# B&R Automation Studio project NAELD004C00R10L518F00 (part 38)

#### Act_Background.st - Change By Project
```iecst
(** 2019-01-08 **)
ACTION Act_Background:

	//Resetting Physical Output
	memset(ADR(a_bPhysicalDO), 0, SIZEOF(a_bPhysicalDO));

	//Digital Output Mapping Physical Output With Config
	IF p_tyDOSettings.diSafetyRlyRst > 0 AND p_tyDOSettings.diSafetyRlyRst <= UDINT_TO_DINT(p_udiMax) THEN
		a_bPhysicalDO[p_tyDOSettings.diSafetyRlyRst]	:= p_bSafetyRlyRst;
	END_IF

	IF p_tyDOSettings.diTLRed > 0 AND p_tyDOSettings.diTLRed <= UDINT_TO_DINT(p_udiMax) THEN
		a_bPhysicalDO[p_tyDOSettings.diTLRed]	:= p_bTLRed;
	END_IF

	IF p_tyDOSettings.diTLAmber > 0 AND p_tyDOSettings.diTLAmber <= UDINT_TO_DINT(p_udiMax) THEN
		a_bPhysicalDO[p_tyDOSettings.diTLAmber]	:= p_bTLAmber;
	END_IF

	IF p_tyDOSettings.diTLGreen > 0 AND p_tyDOSettings.diTLGreen <= UDINT_TO_DINT(p_udiMax) THEN
		a_bPhysicalDO[p_tyDOSettings.diTLGreen]	:= p_bTLGreen;
	END_IF

	IF p_tyDOSettings.diBuzzer > 0 AND p_tyDOSettings.diBuzzer <= UDINT_TO_DINT(p_udiMax) THEN
		a_bPhysicalDO[p_tyDOSettings.diBuzzer]	:= p_bBuzzer;
	END_IF

	IF p_tyDOSettings.diDBAA > 0 AND p_tyDOSettings.diDBAA <= UDINT_TO_DINT(p_udiMax) THEN
		a_bPhysicalDO[p_tyDOSettings.diDBAA]	:= p_bDBAA;
	END_IF

	IF p_tyDOSettings.diDBAB > 0 AND p_tyDOSettings.diDBAB <= UDINT_TO_DINT(p_udiMax) THEN
		a_bPhysicalDO[p_tyDOSettings.diDBAB]	:= p_bDBAB;
	END_IF

	IF p_tyDOSettings.diPullerExtCtrl > 0 AND p_tyDOSettings.diPullerExtCtrl <= UDINT_TO_DINT(p_udiMax) THEN
		a_bPhysicalDO[p_tyDOSettings.diPullerExtCtrl]	:= p_bPullerExtCtrl;
	END_IF

	IF p_tyDOSettings.diPullerRetCtrl > 0 AND p_tyDOSettings.diPullerRetCtrl <= UDINT_TO_DINT(p_udiMax) THEN
		a_bPhysicalDO[p_tyDOSettings.diPullerRetCtrl]	:= p_bPullerRetCtrl;
	END_IF

	IF p_tyDOSettings.diRotPullerCtrl > 0 AND p_tyDOSettings.diRotPullerCtrl <= UDINT_TO_DINT(p_udiMax) THEN
		a_bPhysicalDO[p_tyDOSettings.diRotPullerCtrl]	:= p_bRotPullerCtrl;
	END_IF

	IF p_tyDOSettings.diMag1FixedClampCtrl > 0 AND p_tyDOSettings.diMag1FixedClampCtrl <= UDINT_TO_DINT(p_udiMax) THEN
		a_bPhysicalDO[p_tyDOSettings.diMag1FixedClampCtrl]	:= p_bMag1FixedClampCtrl;
	END_IF

	IF p_tyDOSettings.diMag1RemoteClampCtrl > 0 AND p_tyDOSettings.diMag1RemoteClampCtrl <= UDINT_TO_DINT(p_udiMax) THEN
		a_bPhysicalDO[p_tyDOSettings.diMag1RemoteClampCtrl]	:= p_bMag1RemoteClampCtrl;
	END_IF

	IF p_tyDOSettings.diMag2FixedClampCtrl > 0 AND p_tyDOSettings.diMag2FixedClampCtrl <= UDINT_TO_DINT(p_udiMax) THEN
		a_bPhysicalDO[p_tyDOSettings.diMag2FixedClampCtrl]	:= p_bMag2FixedClampCtrl;
	END_IF

	IF p_tyDOSettings.diMag2RemoteClampCtrl > 0 AND p_tyDOSettings.diMag2RemoteClampCtrl <= UDINT_TO_DINT(p_udiMax) THEN
		a_bPhysicalDO[p_tyDOSettings.diMag2RemoteClampCtrl]	:= p_bMag2RemoteClampCtrl;
	END_IF

	IF p_tyDOSettings.diMag3FixedClampCtrl > 0 AND p_tyDOSettings.diMag3FixedClampCtrl <= UDINT_TO_DINT(p_udiMax) THEN
		a_bPhysicalDO[p_tyDOSettings.diMag3FixedClampCtrl]	:= p_bMag3FixedClampCtrl;
	END_IF

	IF p_tyDOSettings.diMag3RemoteClampCtrl > 0 AND p_tyDOSettings.diMag3RemoteClampCtrl <= UDINT_TO_DINT(p_udiMax) THEN
		a_bPhysicalDO[p_tyDOSettings.diMag3RemoteClampCtrl]	:= p_bMag3RemoteClampCtrl;
	END_IF

	IF p_tyDOSettings.diMag4FixedClampCtrl > 0 AND p_tyDOSettings.diMag4FixedClampCtrl <= UDINT_TO_DINT(p_udiMax) THEN
		a_bPhysicalDO[p_tyDOSettings.diMag4FixedClampCtrl]	:= p_bMag4FixedClampCtrl;
	END_IF

	IF p_tyDOSettings.diMag4RemoteClampCtrl > 0 AND p_tyDOSettings.diMag4RemoteClampCtrl <= UDINT_TO_DINT(p_udiMax) THEN
		a_bPhysicalDO[p_tyDOSettings.diMag4RemoteClampCtrl]	:= p_bMag4RemoteClampCtrl;
	END_IF

		//open clamp control (new)
	IF p_tyDOSettings.diMag1FixedClampOpenCtrl > 0 AND p_tyDOSettings.diMag1FixedClampOpenCtrl <= UDINT_TO_DINT(p_udiMax) THEN
		a_bPhysicalDO[p_tyDOSettings.diMag1FixedClampOpenCtrl]	:= NOT p_bMag1FixedClampOpenCtrl;
	END_IF

	IF p_tyDOSettings.diMag1RemoteClampOpenCtrl > 0 AND p_tyDOSettings.diMag1RemoteClampOpenCtrl <= UDINT_TO_DINT(p_udiMax) THEN
		a_bPhysicalDO[p_tyDOSettings.diMag1RemoteClampOpenCtrl]	:= NOT p_bMag1RemoteClampOpenCtrl;
	END_IF

	IF p_tyDOSettings.diMag2FixedClampOpenCtrl > 0 AND p_tyDOSettings.diMag2FixedClampOpenCtrl <= UDINT_TO_DINT(p_udiMax) THEN
		a_bPhysicalDO[p_tyDOSettings.diMag2FixedClampOpenCtrl]	:= NOT p_bMag2FixedClampOpenCtrl;
	END_IF

	IF p_tyDOSettings.diMag2RemoteClampOpenCtrl > 0 AND p_tyDOSettings.diMag2RemoteClampOpenCtrl <= UDINT_TO_DINT(p_udiMax) THEN
		a_bPhysicalDO[p_tyDOSettings.diMag2RemoteClampOpenCtrl]	:= NOT p_bMag2RemoteClampOpenCtrl;
	END_IF

	IF p_tyDOSettings.diMag3FixedClampOpenCtrl > 0 AND p_tyDOSettings.diMag3FixedClampOpenCtrl <= UDINT_TO_DINT(p_udiMax) THEN
		a_bPhysicalDO[p_tyDOSettings.diMag3FixedClampOpenCtrl]	:= NOT p_bMag3FixedClampOpenCtrl;
	END_IF

	IF p_tyDOSettings.diMag3RemoteClampOpenCtrl > 0 AND p_tyDOSettings.diMag3RemoteClampOpenCtrl <= UDINT_TO_DINT(p_udiMax) THEN
		a_bPhysicalDO[p_tyDOSettings.diMag3RemoteClampOpenCtrl]	:= NOT p_bMag3RemoteClampOpenCtrl;
	END_IF

	IF bShutterTuning = FALSE THEN

		IF p_tyDOSettings.diInShutterOpenCtrl > 0 AND p_tyDOSettings.diInShutterOpenCtrl <= UDINT_TO_DINT(p_udiMax) THEN
			a_bPhysicalDO[p_tyDOSettings.diInShutterOpenCtrl]	:= p_bInShutterOpenCtrl;
		END_IF

		IF p_tyDOSettings.diInShutterCloseCtrl > 0 AND p_tyDOSettings.diInShutterCloseCtrl <= UDINT_TO_DINT(p_udiMax) THEN
			a_bPhysicalDO[p_tyDOSettings.diInShutterCloseCtrl]	:= p_bInShutterCloseCtrl;
		END_IF

		IF p_tyDOSettings.diInShutterOpenCtrl2 > 0 AND p_tyDOSettings.diInShutterOpenCtrl2 <= UDINT_TO_DINT(p_udiMax) THEN
			a_bPhysicalDO[p_tyDOSettings.diInShutterOpenCtrl2]	:= p_bInShutterOpenCtrl2;
		END_IF

		IF p_tyDOSettings.diInShutterCloseCtrl2 > 0 AND p_tyDOSettings.diInShutterCloseCtrl2 <= UDINT_TO_DINT(p_udiMax) THEN
			a_bPhysicalDO[p_tyDOSettings.diInShutterCloseCtrl2]	:= p_bInShutterCloseCtrl2;
		END_IF

		IF p_tyDOSettings.diInShutterOpenCtrl3 > 0 AND p_tyDOSettings.diInShutterOpenCtrl3 <= UDINT_TO_DINT(p_udiMax) THEN
			a_bPhysicalDO[p_tyDOSettings.diInShutterOpenCtrl3]	:= p_bInShutterOpenCtrl3;
		END_IF

		IF p_tyDOSettings.diInShutterCloseCtrl3 > 0 AND p_tyDOSettings.diInShutterCloseCtrl3 <= UDINT_TO_DINT(p_udiMax) THEN
			a_bPhysicalDO[p_tyDOSettings.diInShutterCloseCtrl3]	:= p_bInShutterCloseCtrl3;
		END_IF

		IF p_tyDOSettings.diOutShutterOpenCtrl > 0 AND p_tyDOSettings.diOutShutterOpenCtrl <= UDINT_TO_DINT(p_udiMax) THEN
			a_bPhysicalDO[p_tyDOSettings.diOutShutterOpenCtrl]	:= p_bOutShutterOpenCtrl;
		END_IF

		IF p_tyDOSettings.diOutShutterCloseCtrl > 0 AND p_tyDOSettings.diOutShutterCloseCtrl <= UDINT_TO_DINT(p_udiMax) THEN
			a_bPhysicalDO[p_tyDOSettings.diOutShutterCloseCtrl]	:= p_bOutShutterCloseCtrl;
		END_IF

		IF p_tyDOSettings.diOutShutterOpenCtrl2 > 0 AND p_tyDOSettings.diOutShutterOpenCtrl2 <= UDINT_TO_DINT(p_udiMax) THEN
			a_bPhysicalDO[p_tyDOSettings.diOutShutterOpenCtrl2]	:= p_bOutShutterOpenCtrl2;
		END_IF

		IF p_tyDOSettings.diOutShutterCloseCtrl2 > 0 AND p_tyDOSettings.diOutShutterCloseCtrl2 <= UDINT_TO_DINT(p_udiMax) THEN
			a_bPhysicalDO[p_tyDOSettings.diOutShutterCloseCtrl2]	:= p_bOutShutterCloseCtrl2;
		END_IF

	ELSE

		CASE usiShutterTuningStep OF
			0:
				a_bPhysicalDO[p_tyDOSettings.diInShutterOpenCtrl]	:= TRUE;
				a_bPhysicalDO[p_tyDOSettings.diOutShutterOpenCtrl]	:= TRUE;
				a_bPhysicalDO[p_tyDOSettings.diInShutterOpenCtrl2]	:= TRUE;
				a_bPhysicalDO[p_tyDOSettings.diInShutterOpenCtrl3]	:= TRUE;

				fbShutterTuneOpnTim(IN:= TRUE);
				IF fbShutterTuneOpnTim.Q THEN
					usiShutterTuningStep := 10;
					fbShutterTuneOpnTim(IN:= FALSE);
					a_bPhysicalDO[p_tyDOSettings.diInShutterOpenCtrl]	:= FALSE;
					a_bPhysicalDO[p_tyDOSettings.diOutShutterOpenCtrl]	:= FALSE;
					a_bPhysicalDO[p_tyDOSettings.diInShutterOpenCtrl2]	:= FALSE;
					a_bPhysicalDO[p_tyDOSettings.diInShutterOpenCtrl3]	:= FALSE;
				END_IF
			10:

				a_bPhysicalDO[p_tyDOSettings.diInShutterCloseCtrl]	:= TRUE;
				a_bPhysicalDO[p_tyDOSettings.diOutShutterCloseCtrl]	:= TRUE;
				a_bPhysicalDO[p_tyDOSettings.diInShutterCloseCtrl2]	:= TRUE;
				a_bPhysicalDO[p_tyDOSettings.diInShutterCloseCtrl3]	:= TRUE;

				fbShutterTuneClsTim(IN:= TRUE);
				IF fbShutterTuneClsTim.Q THEN
					usiShutterTuningStep := 0;
					fbShutterTuneClsTim(IN:= FALSE);
					a_bPhysicalDO[p_tyDOSettings.diInShutterCloseCtrl]	:= FALSE;
					a_bPhysicalDO[p_tyDOSettings.diOutShutterCloseCtrl]	:= FALSE;
					a_bPhysicalDO[p_tyDOSettings.diInShutterCloseCtrl2]	:= FALSE;
					a_bPhysicalDO[p_tyDOSettings.diInShutterCloseCtrl3]	:= FALSE;
				END_IF

		END_CASE
	END_IF

	IF p_tyDOSettings.diMag1ConvMtrIn > 0 AND p_tyDOSettings.diMag1ConvMtrIn <= UDINT_TO_DINT(p_udiMax) THEN
		a_bPhysicalDO[p_tyDOSettings.diMag1ConvMtrIn]	:= p_bMag1ConvMtrIn;
	END_IF

	IF p_tyDOSettings.diMag1ConvMtrOut > 0 AND p_tyDOSettings.diMag1ConvMtrOut <= UDINT_TO_DINT(p_udiMax) THEN
		a_bPhysicalDO[p_tyDOSettings.diMag1ConvMtrOut]	:= p_bMag1ConvMtrOut;
	END_IF

	IF p_tyDOSettings.diMag2ConvMtrIn > 0 AND p_tyDOSettings.diMag2ConvMtrIn <= UDINT_TO_DINT(p_udiMax) THEN
		a_bPhysicalDO[p_tyDOSettings.diMag2ConvMtrIn]	:= p_bMag2ConvMtrIn;
	END_IF

	IF p_tyDOSettings.diMag2ConvMtrOut > 0 AND p_tyDOSettings.diMag2ConvMtrOut <= UDINT_TO_DINT(p_udiMax) THEN
		a_bPhysicalDO[p_tyDOSettings.diMag2ConvMtrOut]	:= p_bMag2ConvMtrOut;
	END_IF

	IF p_tyDOSettings.diMag3ConvMtrIn > 0 AND p_tyDOSettings.diMag3ConvMtrIn <= UDINT_TO_DINT(p_udiMax) THEN
		a_bPhysicalDO[p_tyDOSettings.diMag3ConvMtrIn]	:= p_bMag3ConvMtrIn;
	END_IF

	IF p_tyDOSettings.diMag3ConvMtrOut > 0 AND p_tyDOSettings.diMag3ConvMtrOut <= UDINT_TO_DINT(p_udiMax) THEN
		a_bPhysicalDO[p_tyDOSettings.diMag3ConvMtrOut]	:= p_bMag3ConvMtrOut;
	END_IF

	IF p_tyDOSettings.diMag4ConvMtrIn > 0 AND p_tyDOSettings.diMag4ConvMtrIn <= UDINT_TO_DINT(p_udiMax) THEN
		a_bPhysicalDO[p_tyDOSettings.diMag4ConvMtrIn]	:= p_bMag4ConvMtrIn;
	END_IF

	IF p_tyDOSettings.diMag4ConvMtrOut > 0 AND p_tyDOSettings.diMag4ConvMtrOut <= UDINT_TO_DINT(p_udiMax) THEN
		a_bPhysicalDO[p_tyDOSettings.diMag4ConvMtrOut]	:= p_bMag4ConvMtrOut;
	END_IF

	IF p_tyDOSettings.diPullConvMtrOn > 0 AND p_tyDOSettings.diPullConvMtrOn <= UDINT_TO_DINT(p_udiMax) THEN
		a_bPhysicalDO[p_tyDOSettings.diPullConvMtrOn]	:= p_bPullConvMtrOn;
	END_IF

	IF p_tyDOSettings.diMag1SelClampCtrl > 0 AND p_tyDOSettings.diMag1SelClampCtrl <= UDINT_TO_DINT(p_udiMax) THEN
		a_bPhysicalDO[p_tyDOSettings.diMag1SelClampCtrl]	:= p_bMag1SelClampCtrl;
	END_IF

	IF p_tyDOSettings.diMag2SelClampCtrl > 0 AND p_tyDOSettings.diMag2SelClampCtrl <= UDINT_TO_DINT(p_udiMax) THEN
		a_bPhysicalDO[p_tyDOSettings.diMag2SelClampCtrl]	:= p_bMag2SelClampCtrl;
	END_IF

	IF p_tyDOSettings.diMag3SelClampCtrl > 0 AND p_tyDOSettings.diMag3SelClampCtrl <= UDINT_TO_DINT(p_udiMax) THEN
		a_bPhysicalDO[p_tyDOSettings.diMag3SelClampCtrl]	:= p_bMag3SelClampCtrl;
	END_IF

	IF p_tyDOSettings.diMag4SelClampCtrl > 0 AND p_tyDOSettings.diMag4SelClampCtrl <= UDINT_TO_DINT(p_udiMax) THEN
		a_bPhysicalDO[p_tyDOSettings.diMag4SelClampCtrl]	:= p_bMag4SelClampCtrl;
	END_IF

	IF bAgvComIODisabled = FALSE THEN
		//SOT Configuration
		IF p_tyDOSettings.diSOT1MagError > 0 AND p_tyDOSettings.diSOT1MagError <= UDINT_TO_DINT(p_udiMax) THEN
			a_bPhysicalDO[p_tyDOSettings.diSOT1MagError]				:= p_bSOTMagError1;
		END_IF

		IF p_tyDOSettings.diSOT1MagSizeLarge > 0 AND p_tyDOSettings.diSOT1MagSizeLarge <= UDINT_TO_DINT(p_udiMax) THEN
			a_bPhysicalDO[p_tyDOSettings.diSOT1MagSizeLarge]				:= p_bSOTMagSizeLarge1;
		END_IF

		IF p_tyDOSettings.diSOT1MagReady > 0 AND p_tyDOSettings.diSOT1MagReady <= UDINT_TO_DINT(p_udiMax) THEN
			a_bPhysicalDO[p_tyDOSettings.diSOT1MagReady]				:= p_bSOTMagReady1;
		END_IF

		IF p_tyDOSettings.diSOT1MagAvailable > 0 AND p_tyDOSettings.diSOT1MagAvailable <= UDINT_TO_DINT(p_udiMax) THEN
			a_bPhysicalDO[p_tyDOSettings.diSOT1MagAvailable]				:= p_bSOTMagAvailable1;
		END_IF

		IF p_tyDOSettings.diSOT2MagError > 0 AND p_tyDOSettings.diSOT2MagError <= UDINT_TO_DINT(p_udiMax) THEN
			a_bPhysicalDO[p_tyDOSettings.diSOT2MagError]				:= p_bSOTMagError2;
		END_IF

		IF p_tyDOSettings.diSOT2MagSizeLarge > 0 AND p_tyDOSettings.diSOT2MagSizeLarge <= UDINT_TO_DINT(p_udiMax) THEN
			a_bPhysicalDO[p_tyDOSettings.diSOT2MagSizeLarge]				:= p_bSOTMagSizeLarge2;
		END_IF

		IF p_tyDOSettings.diSOT2MagReady > 0 AND p_tyDOSettings.diSOT2MagReady <= UDINT_TO_DINT(p_udiMax) THEN
			a_bPhysicalDO[p_tyDOSettings.diSOT2MagReady]				:= p_bSOTMagReady2;
		END_IF

		IF p_tyDOSettings.diSOT2MagAvailable > 0 AND p_tyDOSettings.diSOT2MagAvailable <= UDINT_TO_DINT(p_udiMax) THEN
			a_bPhysicalDO[p_tyDOSettings.diSOT2MagAvailable]				:= p_bSOTMagAvailable2;
		END_IF

		IF p_tyDOSettings.diSOT3MagError > 0 AND p_tyDOSettings.diSOT3MagError <= UDINT_TO_DINT(p_udiMax) THEN
			a_bPhysicalDO[p_tyDOSettings.diSOT3MagError]				:= p_bSOTMagError3;
		END_IF

		IF p_tyDOSettings.diSOT3MagSizeLarge > 0 AND p_tyDOSettings.diSOT3MagSizeLarge <= UDINT_TO_DINT(p_udiMax) THEN
			a_bPhysicalDO[p_tyDOSettings.diSOT3MagSizeLarge]				:= p_bSOTMagSizeLarge3;
		END_IF

		IF p_tyDOSettings.diSOT3MagReady > 0 AND p_tyDOSettings.diSOT3MagReady <= UDINT_TO_DINT(p_udiMax) THEN
			a_bPhysicalDO[p_tyDOSettings.diSOT3MagReady]				:= p_bSOTMagReady3;
		END_IF

		IF p_tyDOSettings.diSOT3MagAvailable > 0 AND p_tyDOSettings.diSOT3MagAvailable <= UDINT_TO_DINT(p_udiMax) THEN
			a_bPhysicalDO[p_tyDOSettings.diSOT3MagAvailable]				:= p_bSOTMagAvailable3;
		END_IF

		IF p_tyDOSettings.diSOT4MagError > 0 AND p_tyDOSettings.diSOT4MagError <= UDINT_TO_DINT(p_udiMax) THEN
			a_bPhysicalDO[p_tyDOSettings.diSOT4MagError]				:= p_bSOTMagError4;
		END_IF

		IF p_tyDOSettings.diSOT4MagSizeLarge > 0 AND p_tyDOSettings.diSOT4MagSizeLarge <= UDINT_TO_DINT(p_udiMax) THEN
			a_bPhysicalDO[p_tyDOSettings.diSOT4MagSizeLarge]				:= p_bSOTMagSizeLarge4;
		END_IF

		IF p_tyDOSettings.diSOT4MagReady > 0 AND p_tyDOSettings.diSOT4MagReady <= UDINT_TO_DINT(p_udiMax) THEN
			a_bPhysicalDO[p_tyDOSettings.diSOT4MagReady]				:= p_bSOTMagReady4;
		END_IF

		IF p_tyDOSettings.diSOT4MagAvailable > 0 AND p_tyDOSettings.diSOT4MagAvailable <= UDINT_TO_DINT(p_udiMax) THEN
			a_bPhysicalDO[p_tyDOSettings.diSOT4MagAvailable]				:= p_bSOTMagAvailable4;
		END_IF

	ELSE
		a_bPhysicalDO[p_tyDOSettings.diSOT1MagError] := FALSE;
		a_bPhysicalDO[p_tyDOSettings.diSOT1MagSizeLarge] := FALSE;
		a_bPhysicalDO[p_tyDOSettings.diSOT1MagReady] := FALSE;
		a_bPhysicalDO[p_tyDOSettings.diSOT1MagAvailable] := FALSE;

		a_bPhysicalDO[p_tyDOSettings.diSOT2MagError] := FALSE;
		a_bPhysicalDO[p_tyDOSettings.diSOT2MagSizeLarge] := FALSE;
		a_bPhysicalDO[p_tyDOSettings.diSOT2MagReady] := FALSE;
		a_bPhysicalDO[p_tyDOSettings.diSOT2MagAvailable] := FALSE;

		a_bPhysicalDO[p_tyDOSettings.diSOT2MagError] := FALSE;
		a_bPhysicalDO[p_tyDOSettings.diSOT2MagSizeLarge] := FALSE;
		a_bPhysicalDO[p_tyDOSettings.diSOT2MagReady] := FALSE;
		a_bPhysicalDO[p_tyDOSettings.diSOT2MagAvailable] := FALSE;

		a_bPhysicalDO[p_tyDOSettings.diSOT2MagError] := FALSE;
		a_bPhysicalDO[p_tyDOSettings.diSOT2MagSizeLarge] := FALSE;
		a_bPhysicalDO[p_tyDOSettings.diSOT2MagReady] := FALSE;
		a_bPhysicalDO[p_tyDOSettings.diSOT2MagAvailable] := FALSE;
	END_IF

	IF p_eLinkAGVComProtocol = McSetAGVCommHardIO THEN
		IF p_tyDOSettings.diMag1ReqToBring > 0 AND p_tyDOSettings.diMag1ReqToBring <= UDINT_TO_DINT(p_udiMax) THEN
			a_bPhysicalDO[p_tyDOSettings.diMag1ReqToBring]				:= p_bRequestToBring1;
		END_IF

		IF p_tyDOSettings.diMag1ReqToGet > 0 AND p_tyDOSettings.diMag1ReqToGet <= UDINT_TO_DINT(p_udiMax) THEN
			a_bPhysicalDO[p_tyDOSettings.diMag1ReqToGet]				:= p_bRequestToGet1;
		END_IF

		IF p_tyDOSettings.diMag2ReqToBring > 0 AND p_tyDOSettings.diMag2ReqToBring <= UDINT_TO_DINT(p_udiMax) THEN
			a_bPhysicalDO[p_tyDOSettings.diMag2ReqToBring]				:= p_bRequestToBring2;
		END_IF

		IF p_tyDOSettings.diMag2ReqToGet > 0 AND p_tyDOSettings.diMag2ReqToGet <= UDINT_TO_DINT(p_udiMax) THEN
			a_bPhysicalDO[p_tyDOSettings.diMag2ReqToGet]				:= p_bRequestToGet2;
		END_IF

		IF p_tyDOSettings.diMag3ReqToBring > 0 AND p_tyDOSettings.diMag3ReqToBring <= UDINT_TO_DINT(p_udiMax) THEN
			a_bPhysicalDO[p_tyDOSettings.diMag3ReqToBring]				:= p_bRequestToBring3;
		END_IF

		IF p_tyDOSettings.diMag3ReqToGet > 0 AND p_tyDOSettings.diMag3ReqToGet <= UDINT_TO_DINT(p_udiMax) THEN
			a_bPhysicalDO[p_tyDOSettings.diMag3ReqToGet]				:= p_bRequestToGet3;
		END_IF

		IF p_tyDOSettings.diMag4ReqToBring > 0 AND p_tyDOSettings.diMag4ReqToBring <= UDINT_TO_DINT(p_udiMax) THEN
			a_bPhysicalDO[p_tyDOSettings.diMag4ReqToBring]				:= p_bRequestToBring4;
		END_IF

		IF p_tyDOSettings.diMag4ReqToGet > 0 AND p_tyDOSettings.diMag4ReqToGet <= UDINT_TO_DINT(p_udiMax) THEN
			a_bPhysicalDO[p_tyDOSettings.diMag4ReqToGet]				:= p_bRequestToGet4;
		END_IF
	ELSE
		a_bPhysicalDO[p_tyDOSettings.diMag1ReqToBring] := FALSE;
		a_bPhysicalDO[p_tyDOSettings.diMag1ReqToGet] := FALSE;
		a_bPhysicalDO[p_tyDOSettings.diMag2ReqToBring] := FALSE;
		a_bPhysicalDO[p_tyDOSettings.diMag2ReqToGet] := FALSE;
		a_bPhysicalDO[p_tyDOSettings.diMag3ReqToBring] := FALSE;
		a_bPhysicalDO[p_tyDOSettings.diMag3ReqToGet] := FALSE;
		a_bPhysicalDO[p_tyDOSettings.diMag4ReqToBring] := FALSE;
		a_bPhysicalDO[p_tyDOSettings.diMag4ReqToGet] := FALSE;
	END_IF

	IF p_tyDOSettings.diUSBRun > 0 AND p_tyDOSettings.diUSBRun <= UDINT_TO_DINT(p_udiMax) THEN
		a_bPhysicalDO[p_tyDOSettings.diUSBRun]	:= p_bUSBRun;
	END_IF

	IF p_tyDOSettings.diMtrPshrExt > 0 AND p_tyDOSettings.diMtrPshrExt <= UDINT_TO_DINT(p_udiMax) THEN
		a_bPhysicalDO[p_tyDOSettings.diMtrPshrExt]	:= p_bMtrPshrExt;
	END_IF

	IF p_tyDOSettings.diMtrPshrRet > 0 AND p_tyDOSettings.diMtrPshrRet <= UDINT_TO_DINT(p_udiMax) THEN
		a_bPhysicalDO[p_tyDOSettings.diMtrPshrRet]	:= p_bMtrPshrRet;
	END_IF

	IF p_tyDOSettings.diMtrPshrOn > 0 AND p_tyDOSettings.diMtrPshrOn <= UDINT_TO_DINT(p_udiMax) THEN
		a_bPhysicalDO[p_tyDOSettings.diMtrPshrOn]	:= p_bMtrPshrOn;
	END_IF

	IF p_tyDOSettings.diMtrPshrBrakeRls > 0 AND p_tyDOSettings.diMtrPshrBrakeRls <= UDINT_TO_DINT(p_udiMax) THEN
		a_bPhysicalDO[p_tyDOSettings.diMtrPshrBrakeRls]	:= p_bMtrPshrBrakeRls;
	END_IF

	IF p_tyDOSettings.diMtrPshrSpdBinBit0 > 0 AND p_tyDOSettings.diMtrPshrSpdBinBit0 <= UDINT_TO_DINT(p_udiMax) THEN
		a_bPhysicalDO[p_tyDOSettings.diMtrPshrSpdBinBit0]	:= p_bMtrPshrSpdBinBit0;
	END_IF

	IF p_tyDOSettings.diMtrPshrSpdBinBit1 > 0 AND p_tyDOSettings.diMtrPshrSpdBinBit1 <= UDINT_TO_DINT(p_udiMax) THEN
		a_bPhysicalDO[p_tyDOSettings.diMtrPshrSpdBinBit1]	:= p_bMtrPshrSpdBinBit1;
	END_IF

	IF p_tyDOSettings.diMtrPshrSpdBinBit2 > 0 AND p_tyDOSettings.diMtrPshrSpdBinBit2 <= UDINT_TO_DINT(p_udiMax) THEN
		a_bPhysicalDO[p_tyDOSettings.diMtrPshrSpdBinBit2]	:= p_bMtrPshrSpdBinBit2;
	END_IF

	IF p_tyDOSettings.diMtrPshrAlmRst > 0 AND p_tyDOSettings.diMtrPshrAlmRst <= UDINT_TO_DINT(p_udiMax) THEN
		a_bPhysicalDO[p_tyDOSettings.diMtrPshrAlmRst]	:= p_bMtrPshrAlmRst;
	END_IF

	IF p_tyDOSettings.diMag1SafetyBarRetCtrl > 0 AND p_tyDOSettings.diMag1SafetyBarRetCtrl <= UDINT_TO_DINT(p_udiMax) THEN
		a_bPhysicalDO[p_tyDOSettings.diMag1SafetyBarRetCtrl]	:= p_bMag1SafetyBarRetCtrl;
	END_IF

	IF p_tyDOSettings.diMag2SafetyBarRetCtrl > 0 AND p_tyDOSettings.diMag2SafetyBarRetCtrl <= UDINT_TO_DINT(p_udiMax) THEN
		a_bPhysicalDO[p_tyDOSettings.diMag2SafetyBarRetCtrl]	:= p_bMag2SafetyBarRetCtrl;
	END_IF

	IF p_tyDOSettings.diMag3SafetyBarRetCtrl > 0 AND p_tyDOSettings.diMag3SafetyBarRetCtrl <= UDINT_TO_DINT(p_udiMax) THEN
		a_bPhysicalDO[p_tyDOSettings.diMag3SafetyBarRetCtrl]	:= p_bMag3SafetyBarRetCtrl;
	END_IF

	IF p_tyDOSettings.diBypCurtainSen > 0 AND p_tyDOSettings.diBypCurtainSen <= UDINT_TO_DINT(p_udiMax) THEN
		a_bPhysicalDO[p_tyDOSettings.diBypCurtainSen]	:= p_bBypCurtainSen;
	END_IF

	IF p_tyDOSettings.diRstCurtainSen > 0 AND p_tyDOSettings.diRstCurtainSen <= UDINT_TO_DINT(p_udiMax) THEN
		a_bPhysicalDO[p_tyDOSettings.diRstCurtainSen]	:= p_bRstCurtainSen;
	END_IF

	IF p_tyDOSettings.diBypCurtainSensorPBLED > 0 AND p_tyDOSettings.diBypCurtainSensorPBLED <= UDINT_TO_DINT(p_udiMax) THEN	//JOHN
		a_bPhysicalDO[p_tyDOSettings.diBypCurtainSensorPBLED]	:= p_bBypCurtainPBLED;
	END_IF

	IF p_tyDOSettings.diMcSafetySigToDS > 0 AND p_tyDOSettings.diMcSafetySigToDS <= UDINT_TO_DINT(p_udiMax) THEN	//ADD
		a_bPhysicalDO[p_tyDOSettings.diMcSafetySigToDS]	:= p_bUIMachineSafetySigToDS;
	END_IF

	IF p_tyDOSettings.diTrolleyLckCtrl1 > 0 AND p_tyDOSettings.diTrolleyLckCtrl1 <= UDINT_TO_DINT(p_udiMax) THEN
		a_bPhysicalDO[p_tyDOSettings.diTrolleyLckCtrl1]	:= p_bTrolleyExtCtrl;
	END_IF
	IF p_tyDOSettings.diTrolleyLckCtrl2 > 0 AND p_tyDOSettings.diTrolleyLckCtrl2 <= UDINT_TO_DINT(p_udiMax) THEN
		a_bPhysicalDO[p_tyDOSettings.diTrolleyLckCtrl2]	:= p_bTrolleyExtCtrl2;
	END_IF

	//Update Output
	tyDOutput.bSafetyRlyRst			:= p_bSafetyRlyRst;
	tyDOutput.bTLRed				:= p_bTLRed;
	tyDOutput.bTLAmber				:= p_bTLAmber;
	tyDOutput.bTLGreen				:= p_bTLGreen;
	tyDOutput.bBuzzer				:= p_bBuzzer;
	tyDOutput.bDBAA					:= p_bDBAA;
	tyDOutput.bDBAB					:= p_bDBAB;
	tyDOutput.bPullerExtCtrl		:= p_bPullerExtCtrl;
	tyDOutput.bPullerRetCtrl		:= p_bPullerRetCtrl;
	tyDOutput.bRotPullerCtrl		:= p_bRotPullerCtrl;
	tyDOutput.bMag1FixedClampCtrl	:= p_bMag1FixedClampCtrl;
	tyDOutput.bMag1RemoteClampCtrl	:= p_bMag1RemoteClampCtrl;
	tyDOutput.bMag2FixedClampCtrl	:= p_bMag2FixedClampCtrl;
	tyDOutput.bMag2RemoteClampCtrl	:= p_bMag2RemoteClampCtrl;
	tyDOutput.bMag3FixedClampCtrl	:= p_bMag3FixedClampCtrl;
	tyDOutput.bMag3RemoteClampCtrl	:= p_bMag3RemoteClampCtrl;
	tyDOutput.bMag4FixedClampCtrl	:= p_bMag4FixedClampCtrl;
	tyDOutput.bMag4RemoteClampCtrl	:= p_bMag4RemoteClampCtrl;

	tyDOutput.bMag1FixedClampOpenCtrl  := p_bMag1FixedClampOpenCtrl; //new
	tyDOutput.bMag1RemoteClampOpenCtrl  := p_bMag1RemoteClampOpenCtrl;
	tyDOutput.bMag2FixedClampOpenCtrl  := p_bMag2FixedClampOpenCtrl;
	tyDOutput.bMag2RemoteClampOpenCtrl  := p_bMag2RemoteClampOpenCtrl;
	tyDOutput.bMag3FixedClampOpenCtrl  := p_bMag3FixedClampOpenCtrl;
	tyDOutput.bMag3RemoteClampOpenCtrl  := p_bMag3RemoteClampOpenCtrl;

	tyDOutput.bInShutterOpenCtrl	:= p_bInShutterOpenCtrl;
	tyDOutput.bInShutterCloseCtrl	:= p_bInShutterCloseCtrl;
	tyDOutput.bOutShutterOpenCtrl	:= p_bOutShutterOpenCtrl;
	tyDOutput.bOutShutterCloseCtrl	:= p_bOutShutterCloseCtrl;
	tyDOutput.bMag1ConvMtrIn		:= p_bMag1ConvMtrIn;
	tyDOutput.bMag1ConvMtrOut		:= p_bMag1ConvMtrOut;
	tyDOutput.bMag2ConvMtrIn		:= p_bMag2ConvMtrIn;
	tyDOutput.bMag2ConvMtrOut		:= p_bMag2ConvMtrOut;
	tyDOutput.bMag3ConvMtrIn		:= p_bMag3ConvMtrIn;
	tyDOutput.bMag3ConvMtrOut		:= p_bMag3ConvMtrOut;
	tyDOutput.bMag4ConvMtrIn		:= p_bMag4ConvMtrIn;
	tyDOutput.bMag4ConvMtrOut		:= p_bMag4ConvMtrOut;
	tyDOutput.bPullConvMtrOn		:= p_bPullConvMtrOn;
	tyDOutput.bMag1SelClampCtrl		:= p_bMag1SelClampCtrl;
	tyDOutput.bMag2SelClampCtrl		:= p_bMag2SelClampCtrl;
	tyDOutput.bMag3SelClampCtrl		:= p_bMag3SelClampCtrl;
	tyDOutput.bMag4SelClampCtrl		:= p_bMag4SelClampCtrl;
	tyDOutput.bSOT1MagAvailable		:= p_bSOTMagAvailable1;
	tyDOutput.bSOT2MagAvailable		:= p_bSOTMagAvailable2;
	tyDOutput.bSOT3MagAvailable		:= p_bSOTMagAvailable3;
	tyDOutput.bSOT4MagAvailable		:= p_bSOTMagAvailable4;
	tyDOutput.bSOT1MagError			:= p_bSOTMagError1;
	tyDOutput.bSOT2MagError			:= p_bSOTMagError2;
	tyDOutput.bSOT3MagError			:= p_bSOTMagError3;
	tyDOutput.bSOT4MagError			:= p_bSOTMagError4;
	tyDOutput.bSOT1MagReady			:= p_bSOTMagReady1;
	tyDOutput.bSOT2MagReady			:= p_bSOTMagReady2;
	tyDOutput.bSOT3MagReady			:= p_bSOTMagReady3;
	tyDOutput.bSOT4MagReady			:= p_bSOTMagReady4;
	tyDOutput.bSOT1MagSizeLarge		:= p_bSOTMagSizeLarge1;
	tyDOutput.bSOT2MagSizeLarge		:= p_bSOTMagSizeLarge2;
	tyDOutput.bSOT3MagSizeLarge		:= p_bSOTMagSizeLarge3;
	tyDOutput.bSOT4MagSizeLarge		:= p_bSOTMagSizeLarge4;
	tyDOutput.bMag1ReqToBring		:= a_bPhysicalDO[p_tyDOSettings.diMag1ReqToBring];
	tyDOutput.bMag1ReqToGet			:= a_bPhysicalDO[p_tyDOSettings.diMag1ReqToGet];
	tyDOutput.bMag2ReqToBring		:= a_bPhysicalDO[p_tyDOSettings.diMag2ReqToBring];
	tyDOutput.bMag2ReqToGet			:= a_bPhysicalDO[p_tyDOSettings.diMag2ReqToGet];
	tyDOutput.bMag3ReqToBring		:= a_bPhysicalDO[p_tyDOSettings.diMag3ReqToBring];
	tyDOutput.bMag3ReqToGet			:= a_bPhysicalDO[p_tyDOSettings.diMag3ReqToGet];
	tyDOutput.bMag4ReqToBring		:= a_bPhysicalDO[p_tyDOSettings.diMag4ReqToBring];
	tyDOutput.bMag4ReqToGet			:= a_bPhysicalDO[p_tyDOSettings.diMag4ReqToGet];
	tyDOutput.bUSBRun				:= p_bUSBRun;
	tyDOutput.bBypCurtainSen		:= p_bBypCurtainSen;
	tyDOutput.bRstCurtainSen		:= p_bRstCurtainSen;
	tyDOutput.bInShutterOpenCtrl2	:= p_bInShutterOpenCtrl2;
	tyDOutput.bInShutterCloseCtrl2	:= p_bInShutterCloseCtrl2;
	tyDOutput.bInShutterOpenCtrl3	:= p_bInShutterOpenCtrl3;
	tyDOutput.bInShutterCloseCtrl3	:= p_bInShutterCloseCtrl3;
	tyDOutput.bMcSafetySigToDS		:= p_bUIMachineSafetySigToDS;
	tyDOutput.bOutShutterOpenCtrl2	:= p_bOutShutterOpenCtrl2;
	tyDOutput.bOutShutterCloseCtrl2	:= p_bOutShutterCloseCtrl2;

END_ACTION
```

#### InputRef.var - Change By Project
```iecst
(*2019-05-20*)
(**)
(*General*)
VAR
	p_eAct : REFERENCE TO eDOAction;
	p_udiMax : REFERENCE TO UDINT;
END_VAR
(**)
(*Configuration*)
VAR
	p_tyDOSettings : REFERENCE TO tyDigitalOutputSettings;
END_VAR
(**)
VAR
	p_bManual : REFERENCE TO BOOL;
	p_bSafetyRlyRst : REFERENCE TO BOOL;
	p_bTLRed : REFERENCE TO BOOL;
	p_bTLAmber : REFERENCE TO BOOL;
	p_bTLGreen : REFERENCE TO BOOL;
	p_bBuzzer : REFERENCE TO BOOL;
	p_bDBAA : REFERENCE TO BOOL;
	p_bDBAB : REFERENCE TO BOOL;
	p_bPullerExtCtrl : REFERENCE TO BOOL;
	p_bPullerRetCtrl : REFERENCE TO BOOL;
	p_bRotPullerCtrl : REFERENCE TO BOOL;
	p_bMag1SelClampCtrl : REFERENCE TO BOOL;
	p_bMag2SelClampCtrl : REFERENCE TO BOOL;
	p_bMag3SelClampCtrl : REFERENCE TO BOOL;
	p_bMag4SelClampCtrl : REFERENCE TO BOOL;
	p_bMag1FixedClampCtrl : REFERENCE TO BOOL;
	p_bMag1RemoteClampCtrl : REFERENCE TO BOOL;
	p_bMag2FixedClampCtrl : REFERENCE TO BOOL;
	p_bMag2RemoteClampCtrl : REFERENCE TO BOOL;
	p_bMag3FixedClampCtrl : REFERENCE TO BOOL;
	p_bMag3RemoteClampCtrl : REFERENCE TO BOOL;
	p_bMag4FixedClampCtrl : REFERENCE TO BOOL;
	p_bMag4RemoteClampCtrl : REFERENCE TO BOOL;
	p_bInShutterOpenCtrl : REFERENCE TO BOOL;
	p_bInShutterOpenCtrl2 : REFERENCE TO BOOL;
	p_bInShutterOpenCtrl3 : REFERENCE TO BOOL;
	p_bInShutterCloseCtrl : REFERENCE TO BOOL;
	p_bInShutterCloseCtrl2 : REFERENCE TO BOOL;
	p_bInShutterCloseCtrl3 : REFERENCE TO BOOL;
	p_bOutShutterOpenCtrl : REFERENCE TO BOOL;
	p_bOutShutterCloseCtrl : REFERENCE TO BOOL;
	p_bOutShutterOpenCtrl2 : REFERENCE TO BOOL;
	p_bOutShutterCloseCtrl2 : REFERENCE TO BOOL;
	p_bMag1ConvMtrIn : REFERENCE TO BOOL;
	p_bMag1ConvMtrOut : REFERENCE TO BOOL;
	p_bMag2ConvMtrIn : REFERENCE TO BOOL;
	p_bMag2ConvMtrOut : REFERENCE TO BOOL;
	p_bMag3ConvMtrIn : REFERENCE TO BOOL;
	p_bMag3ConvMtrOut : REFERENCE TO BOOL;
	p_bMag4ConvMtrIn : REFERENCE TO BOOL;
	p_bMag4ConvMtrOut : REFERENCE TO BOOL;
	p_bPullConvMtrOn : REFERENCE TO BOOL;
	p_bSOTMagError1 : REFERENCE TO BOOL;
	p_bSOTMagSizeLarge1 : REFERENCE TO BOOL;
	p_bSOTMagReady1 : REFERENCE TO BOOL;
	p_bSOTMagAvailable1 : REFERENCE TO BOOL;
	p_bSOTMagError2 : REFERENCE TO BOOL;
	p_bSOTMagSizeLarge2 : REFERENCE TO BOOL;
	p_bSOTMagReady2 : REFERENCE TO BOOL;
	p_bSOTMagAvailable2 : REFERENCE TO BOOL;
	p_bSOTMagError3 : REFERENCE TO BOOL;
	p_bSOTMagSizeLarge3 : REFERENCE TO BOOL;
	p_bSOTMagReady3 : REFERENCE TO BOOL;
	p_bSOTMagAvailable3 : REFERENCE TO BOOL;
	p_bSOTMagError4 : REFERENCE TO BOOL;
	p_bSOTMagSizeLarge4 : REFERENCE TO BOOL;
	p_bSOTMagReady4 : REFERENCE TO BOOL;
	p_bSOTMagAvailable4 : REFERENCE TO BOOL;
	p_bUSBRun : REFERENCE TO BOOL;
	p_bMag1FixedClampOpenCtrl : REFERENCE TO BOOL;
	p_bMag1RemoteClampOpenCtrl : REFERENCE TO BOOL;
	p_bMag2FixedClampOpenCtrl : REFERENCE TO BOOL;
	p_bMag2RemoteClampOpenCtrl : REFERENCE TO BOOL;
	p_bMag3FixedClampOpenCtrl : REFERENCE TO BOOL;
	p_bMag3RemoteClampOpenCtrl : REFERENCE TO BOOL;
END_VAR
(**)
VAR
	p_bRequestToBring1 : REFERENCE TO BOOL;
	p_bRequestToBring2 : REFERENCE TO BOOL;
	p_bRequestToBring3 : REFERENCE TO BOOL;
	p_bRequestToBring4 : REFERENCE TO BOOL;
	p_bRequestToGet1 : REFERENCE TO BOOL;
	p_bRequestToGet2 : REFERENCE TO BOOL;
	p_bRequestToGet3 : REFERENCE TO BOOL;
	p_bRequestToGet4 : REFERENCE TO BOOL;
END_VAR
(**)
VAR
	p_bMtrPshrExt : REFERENCE TO BOOL;
	p_bMtrPshrRet : REFERENCE TO BOOL;
	p_bMtrPshrOn : REFERENCE TO BOOL;
	p_bMtrPshrBrakeRls : REFERENCE TO BOOL;
	p_bMtrPshrSpdBinBit0 : REFERENCE TO BOOL;
	p_bMtrPshrSpdBinBit1 : REFERENCE TO BOOL;
	p_bMtrPshrSpdBinBit2 : REFERENCE TO BOOL;
	p_bMtrPshrAlmRst : REFERENCE TO BOOL;
	p_bMag1SafetyBarRetCtrl : REFERENCE TO BOOL;
	p_bMag2SafetyBarRetCtrl : REFERENCE TO BOOL;
	p_bMag3SafetyBarRetCtrl : REFERENCE TO BOOL;
	p_bTrolleyExtCtrl : REFERENCE TO BOOL;
	p_bTrolleyExtCtrl2 : REFERENCE TO BOOL;
END_VAR
(**)
VAR
	p_bBypCurtainSen : REFERENCE TO BOOL;
	p_bRstCurtainSen : REFERENCE TO BOOL;
	p_bBypCurtainPBLED : REFERENCE TO BOOL;
	p_bUIMachineSafetySigToDS : REFERENCE TO BOOL;
	p_bDIDSUnlockSafetySig : REFERENCE TO BOOL;
END_VAR
```

#### Local.var - Change By Project
```iecst
(*2019-04-30*)
(**)
(*Local Action, State & Status*)
VAR
	eAct : eDOAction := DOActIdle;
	eStat : eDOAction := DOActIdle;
	eStatus : eFBStatus := Idle;
	sStatTxt : STRING[200] := '';
	a_sStatText : ARRAY[0..50] OF STRING[200] := ['Idling','Resetting All Special Output','Turning On Bypass Cover Switch','Turning Off Bypass Cover Switch',47('')];
END_VAR
(**)
(*Local Alarm*)
(**)
(*Local Output*)
VAR
	tyDOutput : tyDigitalOutput;
END_VAR
(**)
(*Local Input*)
VAR
	tyDOSettings : tyDigitalOutputSettings;
END_VAR
(**)
VAR
	bManual : BOOL := FALSE;
	bSafetyRlyRst : BOOL;
	bTLRed : BOOL;
	bTLAmber : BOOL;
	bTLGreen : BOOL;
	bBuzzer : BOOL;
	bDBAA : BOOL;
	bDBAB : BOOL;
	bPullerExtCtrl : BOOL;
	bPullerRetCtrl : BOOL;
	bRotPullerCtrl : BOOL;
	bMag1FixedClampCtrl : BOOL;
	bMag1RemoteClampCtrl : BOOL;
	bMag2FixedClampCtrl : BOOL;
	bMag2RemoteClampCtrl : BOOL;
	bMag3FixedClampCtrl : BOOL;
	bMag3RemoteClampCtrl : BOOL;
	bMag1FixedClampOpenCtrl : BOOL;
	bMag1RemoteClampOpenCtrl : BOOL;
	bMag2FixedClampOpenCtrl : BOOL;
	bMag2RemoteClampOpenCtrl : BOOL;
	bMag3FixedClampOpenCtrl : BOOL;
	bMag3RemoteClampOpenCtrl : BOOL;
	bInShutterOpenCtrl : BOOL;
	bInShutterCloseCtrl : BOOL;
	bOutShutterOpenCtrl : BOOL;
	bOutShutterCloseCtrl : BOOL;
	bMag1ConvMtrIn : BOOL;
	bMag1ConvMtrOut : BOOL;
	bMag2ConvMtrIn : BOOL;
	bMag2ConvMtrOut : BOOL;
	bMag3ConvMtrIn : BOOL;
	bMag3ConvMtrOut : BOOL;
	bPullConvMtrOn : BOOL;
	bMag1SelClampCtrl : BOOL;
	bMag2SelClampCtrl : BOOL;
	bMag3SelClampCtrl : BOOL;
	bSOTMagError1 : BOOL;
	bSOTMagSLarge1 : BOOL;
	bSOTMagReady1 : BOOL;
	bSOTMagAvailable1 : BOOL;
	bSOTMagError2 : BOOL;
	bSOTMagSLarge2 : BOOL;
	bSOTMagReady2 : BOOL;
	bSOTMagAvailable2 : BOOL;
	bSOTMagError3 : BOOL;
	bSOTMagSLarge3 : BOOL;
	bSOTMagReady3 : BOOL;
	bSOTMagAvailable3 : BOOL;
	bSOTMagError4 : BOOL;
	bSOTMagSLarge4 : BOOL;
	bSOTMagReady4 : BOOL;
	bSOTMagAvailable4 : BOOL;
	bRequestToBring1 : BOOL;
	bRequestToGet1 : BOOL;
	bRequestToBring2 : BOOL;
	bRequestToGet2 : BOOL;
	bRequestToBring3 : BOOL;
	bRequestToGet3 : BOOL;
	bRequestToBring4 : BOOL;
	bRequestToGet4 : BOOL;
	bMag1SafetyBarRetCtrl : BOOL;
	bMag2SafetyBarRetCtrl : BOOL;
	bMag3SafetyBarRetCtrl : BOOL;
	bBypCurtainPBLED : BOOL;
	bBypCurtainSen : BOOL;
	bRstCurtainSen : BOOL;
	bMcSafetySigDS : BOOL;
	bTrolleyExtCtrl : BOOL;
	bTrolleyExtCtrl2 : BOOL;
END_VAR
(**)
(*Local*)
VAR
	bInitDone : BOOL;
	bInitialDone : BOOL;
	a_bPhysicalDO : ARRAY[1..c_udiDOutputMax] OF BOOL;
	eStatOld : eDOAction := DOActIdle;
	usiShutterTuningStep : USINT := 0;
	bShutterTuning : BOOL;
	fbShutterTuneOpnTim : TON := (PT:=T#2s);
	fbShutterTuneClsTim : TON := (PT:=T#2s);
	bAgvComIODisabled : BOOL;
END_VAR
```

### Hermes.var - Change By Project
```iecst
(*2021-08-01*)
(**)
(*Action & State & Status*)
VAR
	p_HermesStat : UDINT;
	p_HermesStatus : UDINT;
	p_HermesStatTxt : UDINT;
	p_HermesMcParamAct : UDINT;
END_VAR
(**)
(*Alarm*)
VAR
	p_HermesAlmData : UDINT;
END_VAR
(**)
(*Output*)
VAR
	p_HermesFileNotFound : UDINT;
	p_HermesConfiguration : UDINT;
	p_HermesConfigurationWr : UDINT;
	p_HermesUSParam1 : UDINT;
	p_HermesUSParam2 : UDINT;
	p_HermesUSParam3 : UDINT;
	p_HermesUSParam4 : UDINT;
	p_HermesDSParam1 : UDINT;
	p_HermesDSParam2 : UDINT;
	p_HermesDSParam3 : UDINT;
	p_HermesDSParam4 : UDINT;
	p_HermesSvyParam : UDINT;
	p_HermesBrdAvlDataTable1stZ : UDINT;
	p_HermesBrdAvlDataTtlIdx1stZ : UDINT;
	p_HermesBrdAvlDataNewBrdAvl1stZ : UDINT;
	p_HermesBrdAvlDataTableLastZ : UDINT;
	p_HermesBrdAvlDataTtlIdxLastZ : UDINT;
	p_HermesBrdAvlDataNewBrdAvlLastZ : UDINT;
	p_HermesBrdId : UDINT;
END_VAR
```

### Program Logical/Hermes/Hermes (IEC) - 1.00.0 - NtHermes v5.00.0 , NtTCP v5.00.0 , NtMessage v5.00.0

#### InputRef.var
```iecst
(*2021-08-01*)
(**)
(*General*)
VAR
	p_eAct : REFERENCE TO eHermesAction;
	p_udiRstErr : REFERENCE TO UDINT;
	p_bPrep : REFERENCE TO BOOL;
	p_bEn : REFERENCE TO BOOL;
	p_bDis : REFERENCE TO BOOL;
END_VAR
(**)
(*Configuration*)
(**)
(*Input*)
VAR
	pa_tyUSParam : REFERENCE TO ARRAY[0..c_diHermesConfigMaxIdx] OF tyHermesUSParam;
	pa_tyDSParam : REFERENCE TO ARRAY[0..c_diHermesConfigMaxIdx] OF tyHermesDSParam;
	p_tyRmtParam : REFERENCE TO tyHermesRmtParam;
	p_tySvyParam : REFERENCE TO tyHermesSvyParam;
	p_sMcId : REFERENCE TO STRING[30];
	p_bRmtHermesWriteConfig : REFERENCE TO BOOL;
	p_bSvyHermesWriteConfig : REFERENCE TO BOOL;
	p_bUISaveHMIConfigure : REFERENCE TO BOOL;
	p_bUISaveHMISvyConfig : REFERENCE TO BOOL;
	p_tyRmtSetConfiguration : REFERENCE TO tyHermesCurrentConfiguration;
	p_bRmtPrep : REFERENCE TO BOOL;
	p_bRmtEn : REFERENCE TO BOOL;
	p_tySvySetConfiguration : REFERENCE TO tyHermesCurrentConfiguration;
	p_bSvyPrep : REFERENCE TO BOOL;
	p_bSvyEn : REFERENCE TO BOOL;
	p_sRetainFileName1 : REFERENCE TO STRING[80];
	p_sRetainFileName2 : REFERENCE TO STRING[80];
	p_sRetainFileName3 : REFERENCE TO STRING[80];
	p_sRetainFileName4 : REFERENCE TO STRING[80];
	p_udiRetainDataAddr1 : REFERENCE TO UDINT;
	p_udiRetainDataLen1 : REFERENCE TO UDINT;
	p_udiRetainDataAddr2 : REFERENCE TO UDINT;
	p_udiRetainDataLen2 : REFERENCE TO UDINT;
	p_udiRetainDataAddr3 : REFERENCE TO UDINT;
	p_udiRetainDataLen3 : REFERENCE TO UDINT;
	p_udiRetainDataAddr4 : REFERENCE TO UDINT;
	p_udiRetainDataLen4 : REFERENCE TO UDINT;
	p_sConfigFileName : REFERENCE TO STRING[80];
	p_sProgNm : REFERENCE TO STRING[15];
	p_bNtSettingsLoadDone : REFERENCE TO BOOL;
END_VAR
(**)
(*RmtHermes*)
VAR
	p_bRmtFoundIndexUS1 : REFERENCE TO BOOL;
	p_bRmtFoundIndexUS2 : REFERENCE TO BOOL;
	p_bRmtFoundIndexUS3 : REFERENCE TO BOOL;
	p_bRmtFoundIndexUS4 : REFERENCE TO BOOL;
	p_bRmtFoundIndexDS1 : REFERENCE TO BOOL;
	p_bRmtFoundIndexDS2 : REFERENCE TO BOOL;
	p_bRmtFoundIndexDS3 : REFERENCE TO BOOL;
	p_bRmtFoundIndexDS4 : REFERENCE TO BOOL;
	p_udiRmtIndexUS1 : REFERENCE TO UDINT;
	p_udiRmtIndexUS2 : REFERENCE TO UDINT;
	p_udiRmtIndexUS3 : REFERENCE TO UDINT;
	p_udiRmtIndexUS4 : REFERENCE TO UDINT;
	p_udiRmtIndexDS1 : REFERENCE TO UDINT;
	p_udiRmtIndexDS2 : REFERENCE TO UDINT;
	p_udiRmtIndexDS3 : REFERENCE TO UDINT;
	p_udiRmtIndexDS4 : REFERENCE TO UDINT;
END_VAR
(**)
(*SvyHermes*)
VAR
	p_bSvyFoundIndexUS1 : REFERENCE TO BOOL;
	p_bSvyFoundIndexUS2 : REFERENCE TO BOOL;
	p_bSvyFoundIndexUS3 : REFERENCE TO BOOL;
	p_bSvyFoundIndexUS4 : REFERENCE TO BOOL;
	p_bSvyFoundIndexDS1 : REFERENCE TO BOOL;
	p_bSvyFoundIndexDS2 : REFERENCE TO BOOL;
	p_bSvyFoundIndexDS3 : REFERENCE TO BOOL;
	p_bSvyFoundIndexDS4 : REFERENCE TO BOOL;
	p_udiSvyIndexUS1 : REFERENCE TO UDINT;
	p_udiSvyIndexUS2 : REFERENCE TO UDINT;
	p_udiSvyIndexUS3 : REFERENCE TO UDINT;
	p_udiSvyIndexUS4 : REFERENCE TO UDINT;
	p_udiSvyIndexDS1 : REFERENCE TO UDINT;
	p_udiSvyIndexDS2 : REFERENCE TO UDINT;
	p_udiSvyIndexDS3 : REFERENCE TO UDINT;
	p_udiSvyIndexDS4 : REFERENCE TO UDINT;
END_VAR
(**)
```

#### InputRef_Link.var
```iecst
(*2021-08-01*)
(**)
VAR
	p_bLinkStartupRun : REFERENCE TO BOOL;
	pa_usiMacAddr : REFERENCE TO ARRAY[0..5] OF USINT;
	p_tyDTStructure : REFERENCE TO DTStructure;
END_VAR
(**)
VAR
	pa_tyLinkXMLTableDataBrdAvl1 : REFERENCE TO ARRAY[0..200] OF tyXMLTableDat;
	p_iLinkXMLTableDataBrdAvlTtlIdx1 : REFERENCE TO INT;
	pa_tyLinkXMLTableDataBrdAvl2 : REFERENCE TO ARRAY[0..200] OF tyXMLTableDat;
	p_iLinkXMLTableDataBrdAvlTtlIdx2 : REFERENCE TO INT;
	pa_tyLinkXMLTableDataBrdAvl3 : REFERENCE TO ARRAY[0..200] OF tyXMLTableDat;
	p_iLinkXMLTableDataBrdAvlTtlIdx3 : REFERENCE TO INT;
	pa_tyLinkXMLTableDataBrdAvl4 : REFERENCE TO ARRAY[0..200] OF tyXMLTableDat;
	p_iLinkXMLTableDataBrdAvlTtlIdx4 : REFERENCE TO INT;
END_VAR
(**)
VAR
	tyHermesBrdAvlData : tyHermesBrdAvlDat;
	a_tyHermesBrdAvlData : ARRAY[1..200] OF tyHermesBrdAvlDat; (*Cater Up to 6 Zones*)
END_VAR
(**)
(*Zone 1*)
VAR
	p_bLinkOpsInitGConv1StepInitDone : REFERENCE TO BOOL;
	p_bLinkOpsInitGConv1MidHvBrd : REFERENCE TO BOOL;
	p_bLinkOpsInitGConv1EndHvBrd : REFERENCE TO BOOL;
	p_bLinkOpsGConv1HvBrd : REFERENCE TO BOOL;
	p_bLinkOpsGConv1StepEntBrd : REFERENCE TO BOOL;
	p_bLinkUSHermesTransporting : REFERENCE TO BOOL;
	p_bLinkUSSMEMATransporting : REFERENCE TO BOOL;
END_VAR
(**)
(*Zone 2*)
VAR
	p_bLinkOpsInitGConv2StepInitDone : REFERENCE TO BOOL;
	p_bLinkOpsInitGConv2MidHvBrd : REFERENCE TO BOOL;
	p_bLinkOpsInitGConv2EndHvBrd : REFERENCE TO BOOL;
	p_bLinkOpsGConv2HvBrd : REFERENCE TO BOOL;
	p_bLinkOpsGConv2StepEntBrd : REFERENCE TO BOOL;
	p_bLinkUSSMEMA2Transporting : REFERENCE TO BOOL;
END_VAR
(**)
```

#### Local.var
```iecst
(*2021-08-01*)
(**)
(*Local Action, State & Status*)
VAR
	eAct : eHermesAction := HermesActIdle;
	eStat : eHermesAction := HermesActIdle;
	eStatus : eFBStatus := Idle;
	udiStatus : UDINT := 0;
	sStatTxt : STRING[200] := '';
	a_sStatText : ARRAY[0..50] OF STRING[200] := ['Idling','Background Starting Operations','Background Stopping Operations','Deleting Old Log File','Creating Directory','Writing Retain File','Reading Retain File','Writing Configuration File','Reading Configuration File',42('')];
END_VAR
(**)
(*Local Alarm*)
VAR
	tyAlmData : tyAlmDat;
	a_tyAlmText : ARRAY[10000..10099] OF tyAlmTxt := [(sAlmText:='Create User Directory Error',sRcyText:='An Error Occurred While Attempting To Create User Directory. Please Contact Nutek For A Possible Solution'),(sAlmText:='Create Retain Directory Error',sRcyText:='An Error Occurred While Attempting To Create Retain Directory. Please Contact Nutek For A Possible Solution'),(sAlmText:='File Open Error While Reading Retain File',sRcyText:='An Error Was Encountered While Trying To Open File. Please Contact Nutek For A Possible Solution.'),(sAlmText:='File Read Error While Reading Retain File',sRcyText:='An Error Was Encountered While Trying To Read File. Please Contact Nutek For A Possible Solution.'),(sAlmText:='File Close Error While Reading Retain File',sRcyText:='An Error Was Encountered While Trying To Close File. Please Contact Nutek For A Possible Solution.'),(sAlmText:='File Open Error While Writing Retain File',sRcyText:='An Error Was Encountered While Trying To Open File. Please Contact Nutek For A Possible Solution.'),(sAlmText:='File Create Error While Writing Retain File',sRcyText:='An Error Was Encountered While Trying To Create File. Please Contact Nutek For A Possible Solution.'),(sAlmText:='File Write Error While Writing Retain File',sRcyText:='An Error Was Encountered While Trying To Write File. Please Contact Nutek For A Possible Solution.'),(sAlmText:='File Close Error While Writing Retain File',sRcyText:='An Error Was Encountered While Trying To Close File. Please Contact Nutek For A Possible Solution.'),(sAlmText:='Directory Does Not Exist While Writing Retain File',sRcyText:='The Directory Does Not Exist. Please Contact Nutek For A Possible Solution.'),(sAlmText:='Create Log Directory Error',sRcyText:='An Error Occurred While Attempting To Create Log Directory. Please Contact Nutek For A Possible Solution'),(sAlmText:='Create Machine Parameter Directory Error',sRcyText:='An Error Occurred While Attempting To Create Machine Parameter Directory. Please Contact Nutek For A Possible Solution'),(sAlmText:='File Open Error While Reading Config File',sRcyText:='An Error Was Encountered While Trying To Open File. Please Contact Nutek For A Possible Solution.'),(sAlmText:='File Read Error While Reading Config File',sRcyText:='An Error Was Encountered While Trying To Read File. Please Contact Nutek For A Possible Solution.'),(sAlmText:='File Close Error While Reading Config File',sRcyText:='An Error Was Encountered While Trying To Close File. Please Contact Nutek For A Possible Solution.'),(sAlmText:='File Open Error While Writing Config File',sRcyText:='An Error Was Encountered While Trying To Open File. Please Contact Nutek For A Possible Solution.'),(sAlmText:='File Create Error While Writing Config File',sRcyText:='An Error Was Encountered While Trying To Create File. Please Contact Nutek For A Possible Solution.'),(sAlmText:='File Write Error While Writing Config File',sRcyText:='An Error Was Encountered While Trying To Write File. Please Contact Nutek For A Possible Solution.'),(sAlmText:='File Close Error While Writing Config File',sRcyText:='An Error Was Encountered While Trying To Close File. Please Contact Nutek For A Possible Solution.'),(sAlmText:='Directory Does Not Exist While Writing Config File',sRcyText:='The Directory Does Not Exist. Please Contact Nutek For A Possible Solution.'),(0),2(0),3((0)),0,3((0)),(sAlmText:='File Open Error While Writing Retain File Lane 2',sRcyText:='An Error Was Encountered While Trying To Open File. Please Contact Nutek For A Possible Solution.'),(0),(sAlmText:='File Open Error While Reading Lane 2 Retain File',sRcyText:='An Error Was Encountered While Trying To Open File. Please Contact Nutek For A Possible Solution.'),(sAlmText:='File Read Error While Reading Lane 2 Retain File',sRcyText:='An Error Was Encountered While Trying To Read File. Please Contact Nutek For A Possible Solution.'),(sAlmText:='File Close Error While Reading Lane 2 Retain File',sRcyText:='An Error Was Encountered While Trying To Close File. Please Contact Nutek For A Possible Solution.'),(sAlmText:='File Open Error While Writing Lane 2 Retain File',sRcyText:='An Error Was Encountered While Trying To Open File. Please Contact Nutek For A Possible Solution.'),(sAlmText:='File Create Error While Writing Lane 2 Retain File',sRcyText:='An Error Was Encountered While Trying To Create File. Please Contact Nutek For A Possible Solution.'),(sAlmText:='File Write Error While Writing Lane 2 Retain File',sRcyText:='An Error Was Encountered While Trying To Write File. Please Contact Nutek For A Possible Solution.'),(sAlmText:='File Close Error While Writing Lane 2 Retain File',sRcyText:='An Error Was Encountered While Trying To Close File. Please Contact Nutek For A Possible Solution.'),(sAlmText:='Directory Does Not Exist While Writing Lane 2 Retain File',sRcyText:='The Directory Does Not Exist. Please Contact Nutek For A Possible Solution.'),2((0)),(sAlmText:='File Open Error While Reading Lane 3 Retain File',sRcyText:='An Error Was Encountered While Trying To Open File. Please Contact Nutek For A Possible Solution.'),(sAlmText:='File Read Error While Reading Lane 3 Retain File',sRcyText:='An Error Was Encountered While Trying To Read File. Please Contact Nutek For A Possible Solution.'),(sAlmText:='File Close Error While Reading Lane 3 Retain File',sRcyText:='An Error Was Encountered While Trying To Close File. Please Contact Nutek For A Possible Solution.'),(sAlmText:='File Open Error While Writing Lane 3 Retain File',sRcyText:='An Error Was Encountered While Trying To Open File. Please Contact Nutek For A Possible Solution.'),(sAlmText:='File Create Error While Writing Lane 3 Retain File',sRcyText:='An Error Was Encountered While Trying To Create File. Please Contact Nutek For A Possible Solution.'),(sAlmText:='File Write Error While Writing Lane 3 Retain File',sRcyText:='An Error Was Encountered While Trying To Write File. Please Contact Nutek For A Possible Solution.'),(sAlmText:='File Close Error While Writing Lane 3 Retain File',sRcyText:='An Error Was Encountered While Trying To Close File. Please Contact Nutek For A Possible Solution.'),(sAlmText:='Directory Does Not Exist While Writing Lane 3 Retain File',sRcyText:='The Directory Does Not Exist. Please Contact Nutek For A Possible Solution.'),2((0)),(sAlmText:='File Open Error While Reading Lane 4 Retain File',sRcyText:='An Error Was Encountered While Trying To Open File. Please Contact Nutek For A Possible Solution.'),(sAlmText:='File Read Error While Reading Lane 4 Retain File',sRcyText:='An Error Was Encountered While Trying To Read File. Please Contact Nutek For A Possible Solution.'),(sAlmText:='File Close Error While Reading Lane 4 Retain File',sRcyText:='An Error Was Encountered While Trying To Close File. Please Contact Nutek For A Possible Solution.'),(sAlmText:='File Open Error While Writing Lane 4 Retain File',sRcyText:='An Error Was Encountered While Trying To Open File. Please Contact Nutek For A Possible Solution.'),(sAlmText:='File Create Error While Writing Lane 4 Retain File',sRcyText:='An Error Was Encountered While Trying To Create File. Please Contact Nutek For A Possible Solution.'),(sAlmText:='File Write Error While Writing Lane 4 Retain File',sRcyText:='An Error Was Encountered While Trying To Write File. Please Contact Nutek For A Possible Solution.'),(sAlmText:='File Close Error While Writing Lane 4 Retain File',sRcyText:='An Error Was Encountered While Trying To Close File. Please Contact Nutek For A Possible Solution.'),(sAlmText:='Directory Does Not Exist While Writing Lane 4 Retain File',sRcyText:='The Directory Does Not Exist. Please Contact Nutek For A Possible Solution.'),40((0))];
END_VAR
(**)
(*Local Output*)
VAR
	bFileNotFound : BOOL;
	tyCurrConfiguration : tyHermesConfiguration := (a_tyUSParam:=[(tSndAlive:=T#60s,iLaneID:=1),3(0)],a_tyDSParam:=[(tSndAlive:=T#60s,uiSvrPort:=502,iLaneID:=1),0,2((0))]);
	tyConfigurationWr : tyHermesConfiguration;
END_VAR
(**)
(*Local Input*)
VAR
	udiRstErr : UDINT := 0;
	bPrep : BOOL := TRUE;
	bEn : BOOL := TRUE;
	bDis : BOOL := FALSE;
	a_tyUSParam : ARRAY[0..c_diHermesConfigMaxIdx] OF tyHermesUSParam;
	a_tyDSParam : ARRAY[0..c_diHermesConfigMaxIdx] OF tyHermesDSParam;
	tyRmtParam : tyHermesRmtParam;
	tySvyParam : tyHermesSvyParam;
	tyRmtSetConfiguration : tyHermesCurrentConfiguration;
	tySvySetConfiguration : tyHermesCurrentConfiguration;
	bRmtPrep : BOOL := FALSE;
	bRmtEn : BOOL := FALSE;
	bSvyPrep : BOOL := FALSE;
	bSvyEn : BOOL := FALSE;
	sRetainFileName1 : STRING[80] := 'HermesLane1.dat';
	sRetainFileName2 : STRING[80] := 'HermesLane2.dat';
	sRetainFileName3 : STRING[80] := 'HermesLane3.dat';
	sRetainFileName4 : STRING[80] := 'HermesLane4.dat';
	udiRetainDataAddr1 : UDINT;
	udiRetainDataLen1 : UDINT;
	udiRetainDataAddr2 : UDINT;
	udiRetainDataLen2 : UDINT;
	udiRetainDataAddr3 : UDINT;
	udiRetainDataLen3 : UDINT;
	udiRetainDataAddr4 : UDINT;
	udiRetainDataLen4 : UDINT;
	sConfigFileName : STRING[80] := 'Hermes.dat';
	sProgNm : STRING[15] := 'Hermes';
	bNtSettingsLoadDone : BOOL := TRUE;
	bRmtHermesWriteConfig : BOOL := TRUE;
	bSvyHermesWriteConfig : BOOL := TRUE;
	bUISaveHMIConfigure : BOOL := TRUE;
	bUISaveHMISvyConfig : BOOL := TRUE;
	sMcId : STRING[30] := '';
	bRmtFoundIndexUS1 : BOOL := FALSE;
	bRmtFoundIndexUS2 : BOOL := FALSE;
	bRmtFoundIndexUS3 : BOOL := FALSE;
	bRmtFoundIndexUS4 : BOOL := FALSE;
	bRmtFoundIndexDS1 : BOOL := FALSE;
	bRmtFoundIndexDS2 : BOOL := FALSE;
	bRmtFoundIndexDS3 : BOOL := FALSE;
	bRmtFoundIndexDS4 : BOOL := FALSE;
	udiRmtIndexUS1 : UDINT := 0;
	udiRmtIndexUS2 : UDINT := 0;
	udiRmtIndexUS3 : UDINT := 0;
	udiRmtIndexUS4 : UDINT := 0;
	udiRmtIndexDS1 : UDINT := 0;
	udiRmtIndexDS2 : UDINT := 0;
	udiRmtIndexDS3 : UDINT := 0;
	udiRmtIndexDS4 : UDINT := 0;
	bSvyFoundIndexUS1 : BOOL := FALSE;
	bSvyFoundIndexUS2 : BOOL := FALSE;
	bSvyFoundIndexUS3 : BOOL := FALSE;
	bSvyFoundIndexUS4 : BOOL := FALSE;
	bSvyFoundIndexDS1 : BOOL := FALSE;
	bSvyFoundIndexDS2 : BOOL := FALSE;
	bSvyFoundIndexDS3 : BOOL := FALSE;
	bSvyFoundIndexDS4 : BOOL := FALSE;
	udiSvyIndexUS1 : UDINT := 0;
	udiSvyIndexUS2 : UDINT := 0;
	udiSvyIndexUS3 : UDINT := 0;
	udiSvyIndexUS4 : UDINT := 0;
	udiSvyIndexDS1 : UDINT := 0;
	udiSvyIndexDS2 : UDINT := 0;
	udiSvyIndexDS3 : UDINT := 0;
	udiSvyIndexDS4 : UDINT := 0;
	sGenBrdUUID : STRING[36];
END_VAR
(**)
(*Local*)
VAR
	bRstErr : BOOL;
	udiRstErrOld : UDINT;
	bInitDone : BOOL;
	bInitialDone : BOOL;
	bHermesWriteRetainLane1 : BOOL;
	bHermesWriteRetainLane2 : BOOL;
	bHermesWriteRetainLane3 : BOOL;
	bHermesWriteRetainLane4 : BOOL;
	usiStep : USINT;
	tyConfigurationHMI : tyHermesConfiguration;
	eStatOld : eHermesAction := HermesActIdle;
	fbDirCreate1 : fbDirCreate;
	fbDirCreate2 : fbDirCreate;
	fbDirCreate3 : fbDirCreate;
	fbDirCreate4 : fbDirCreate;
	fbFileRead1 : fbFileFullRead;
	fbFileWrite1 : fbFileFullWrite;
	fbFileRead2 : fbFileFullRead;
	fbFileWrite2 : fbFileFullWrite;
	fbFileRead3 : fbFileFullRead;
	fbFileWrite3 : fbFileFullWrite;
	fbFileRead4 : fbFileFullRead;
	fbFileWrite4 : fbFileFullWrite;
	fbFileRead5 : fbFileFullRead;
	fbFileWrite5 : fbFileFullWrite;
	i : INT;
	udiModuleNum : UDINT := 2901;
END_VAR
```

#### Act_Alarm.st
```iecst
(** 2021-08-01 **)
ACTION Act_Alarm:

	//Error
	IF EDGEPOS(eStatus = Error) THEN

		tyAlmData.sProgNm		:= p_sProgNm;
		tyAlmData.udiCode		:= udiStatus;
		tyAlmData.eSeverity		:= AlmSeverityError;
		tyAlmData.udiRunTime	:= tyAlmData.udiRunTime + 1;
		tyAlmData.bAlm			:= TRUE;
		tyAlmData.udiModuleNum  := udiModuleNum;
		g_sHermesProgNm		:= p_sProgNm;
		//Get Error Message
		IF tyAlmData.udiCode < 10000 OR tyAlmData.udiCode > 10099 THEN
			tyAlmData.sAlmMsg	:= 'Unknown';
			tyAlmData.sRcyMsg	:= 'Unknown';
		ELSE
			tyAlmData.sAlmMsg	:= a_tyAlmText[tyAlmData.udiCode].sAlmText;
			tyAlmData.sRcyMsg	:= a_tyAlmText[tyAlmData.udiCode].sRcyText;
		END_IF

		sStatTxt	:= tyAlmData.sAlmMsg;

	ELSIF bRstErr AND (tyAlmData.udiCode <> 0) THEN

		tyAlmData.udiCode	:= 0;
		tyAlmData.eSeverity	:= AlmSeverityNA;
		tyAlmData.sAlmMsg	:= '';
		tyAlmData.sRcyMsg	:= '';
		tyAlmData.bAlm			:= FALSE;
		sStatTxt	:= a_sStatText[eStat];

	END_IF

END_ACTION
```

#### Act_Background.st
```iecst
(** 2021-08-01 **)
ACTION Act_Background:

	//Update Configuration

	IF p_bSvyPrep = TRUE AND p_bSvyEn = TRUE AND p_bSvyHermesWriteConfig THEN

		IF p_bSvyFoundIndexUS1 THEN
			tyConfigurationWr.a_tyUSParam[0].iLaneID		            := p_tySvySetConfiguration.tyData.a_tyUpstreamConfigurations[p_udiSvyIndexUS1].iUpstreamLaneId;
			tyConfigurationWr.a_tyUSParam[0].sHostAddress           	:= p_tySvySetConfiguration.tyData.a_tyUpstreamConfigurations[p_udiSvyIndexUS1].sHostAddress;
			tyConfigurationWr.a_tyUSParam[0].uiHostPort	                := p_tySvySetConfiguration.tyData.a_tyUpstreamConfigurations[p_udiSvyIndexUS1].uiPort;
			tyConfigurationWr.a_tyUSParam[0].sUpstreamInterfaceId   	:= p_tySvySetConfiguration.tyData.a_tyUpstreamConfigurations[p_udiSvyIndexUS1].sUpstreamInterfaceId;
		END_IF

		IF p_bSvyFoundIndexUS2 THEN
			tyConfigurationWr.a_tyUSParam[1].iLaneID		            := p_tySvySetConfiguration.tyData.a_tyUpstreamConfigurations[p_udiSvyIndexUS2].iUpstreamLaneId;
			tyConfigurationWr.a_tyUSParam[1].sHostAddress           	:= p_tySvySetConfiguration.tyData.a_tyUpstreamConfigurations[p_udiSvyIndexUS2].sHostAddress;
			tyConfigurationWr.a_tyUSParam[1].uiHostPort	                := p_tySvySetConfiguration.tyData.a_tyUpstreamConfigurations[p_udiSvyIndexUS2].uiPort;
			tyConfigurationWr.a_tyUSParam[1].sUpstreamInterfaceId   	:= p_tySvySetConfiguration.tyData.a_tyUpstreamConfigurations[p_udiSvyIndexUS2].sUpstreamInterfaceId;
		END_IF

		IF p_bSvyFoundIndexUS3 THEN
			tyConfigurationWr.a_tyUSParam[2].iLaneID		            := p_tySvySetConfiguration.tyData.a_tyUpstreamConfigurations[p_udiSvyIndexUS3].iUpstreamLaneId;
			tyConfigurationWr.a_tyUSParam[2].sHostAddress           	:= p_tySvySetConfiguration.tyData.a_tyUpstreamConfigurations[p_udiSvyIndexUS3].sHostAddress;
			tyConfigurationWr.a_tyUSParam[2].uiHostPort	                := p_tySvySetConfiguration.tyData.a_tyUpstreamConfigurations[p_udiSvyIndexUS3].uiPort;
			tyConfigurationWr.a_tyUSParam[2].sUpstreamInterfaceId   	:= p_tySvySetConfiguration.tyData.a_tyUpstreamConfigurations[p_udiSvyIndexUS3].sUpstreamInterfaceId;
		END_IF

		IF p_bSvyFoundIndexUS4 THEN
			tyConfigurationWr.a_tyUSParam[3].iLaneID		            := p_tySvySetConfiguration.tyData.a_tyUpstreamConfigurations[p_udiSvyIndexUS4].iUpstreamLaneId;
			tyConfigurationWr.a_tyUSParam[3].sHostAddress           	:= p_tySvySetConfiguration.tyData.a_tyUpstreamConfigurations[p_udiSvyIndexUS4].sHostAddress;
			tyConfigurationWr.a_tyUSParam[3].uiHostPort	                := p_tySvySetConfiguration.tyData.a_tyUpstreamConfigurations[p_udiSvyIndexUS4].uiPort;
			tyConfigurationWr.a_tyUSParam[3].sUpstreamInterfaceId   	:= p_tySvySetConfiguration.tyData.a_tyUpstreamConfigurations[p_udiSvyIndexUS4].sUpstreamInterfaceId;
		END_IF

		IF p_bSvyFoundIndexDS1 THEN
			tyConfigurationWr.a_tyDSParam[0].iLaneID	            	:= p_tySvySetConfiguration.tyData.a_tyDownstreamConfigurations[p_udiSvyIndexDS1].iDownstreamLaneId;
			tyConfigurationWr.a_tyDSParam[0].uiSvrPort               	:= p_tySvySetConfiguration.tyData.a_tyDownstreamConfigurations[p_udiSvyIndexDS1].uiPort;
			tyConfigurationWr.a_tyDSParam[0].sDownstreamInterfaceId  	:= p_tySvySetConfiguration.tyData.a_tyDownstreamConfigurations[p_udiSvyIndexDS1].sDownstreamInterfaceId;
		END_IF

		IF p_bSvyFoundIndexDS2 THEN
			tyConfigurationWr.a_tyDSParam[1].iLaneID	            	:= p_tySvySetConfiguration.tyData.a_tyDownstreamConfigurations[p_udiSvyIndexDS2].iDownstreamLaneId;
			tyConfigurationWr.a_tyDSParam[1].uiSvrPort               	:= p_tySvySetConfiguration.tyData.a_tyDownstreamConfigurations[p_udiSvyIndexDS2].uiPort;
			tyConfigurationWr.a_tyDSParam[1].sDownstreamInterfaceId  	:= p_tySvySetConfiguration.tyData.a_tyDownstreamConfigurations[p_udiSvyIndexDS2].sDownstreamInterfaceId;
		END_IF

		IF p_bSvyFoundIndexDS3 THEN
			tyConfigurationWr.a_tyDSParam[2].iLaneID	            	:= p_tySvySetConfiguration.tyData.a_tyDownstreamConfigurations[p_udiSvyIndexDS3].iDownstreamLaneId;
			tyConfigurationWr.a_tyDSParam[2].uiSvrPort               	:= p_tySvySetConfiguration.tyData.a_tyDownstreamConfigurations[p_udiSvyIndexDS3].uiPort;
			tyConfigurationWr.a_tyDSParam[2].sDownstreamInterfaceId  	:= p_tySvySetConfiguration.tyData.a_tyDownstreamConfigurations[p_udiSvyIndexDS3].sDownstreamInterfaceId;
		END_IF

		IF p_bSvyFoundIndexDS4 THEN
			tyConfigurationWr.a_tyDSParam[3].iLaneID	            	:= p_tySvySetConfiguration.tyData.a_tyDownstreamConfigurations[p_udiSvyIndexDS4].iDownstreamLaneId;
			tyConfigurationWr.a_tyDSParam[3].uiSvrPort               	:= p_tySvySetConfiguration.tyData.a_tyDownstreamConfigurations[p_udiSvyIndexDS4].uiPort;
			tyConfigurationWr.a_tyDSParam[3].sDownstreamInterfaceId  	:= p_tySvySetConfiguration.tyData.a_tyDownstreamConfigurations[p_udiSvyIndexDS4].sDownstreamInterfaceId;
		END_IF

		IF p_tySvySetConfiguration.tyAvl.bMachineId = TRUE THEN

			tyConfigurationWr.a_tyUSParam[0].sMachineId		:= p_tySvySetConfiguration.tyData.sMachineId;
			tyConfigurationWr.a_tyDSParam[0].sMachineId		:= p_tySvySetConfiguration.tyData.sMachineId;
			tyConfigurationWr.tySvyParam.sMachineId		    := p_tySvySetConfiguration.tyData.sMachineId;

		END_IF

		IF p_tySvySetConfiguration.tyAvl.bSupervisorySystemPort = TRUE THEN

			tyConfigurationWr.tySvyParam.uiSvySvstemPort	:= p_tySvySetConfiguration.tyData.uiSupervisorySystemPort;

		END_IF

	ELSIF p_bRmtPrep = TRUE AND p_bRmtEn = TRUE AND p_bRmtHermesWriteConfig THEN

		IF p_bRmtFoundIndexUS1 THEN
			tyConfigurationWr.a_tyUSParam[0].iLaneID		            := p_tyRmtSetConfiguration.tyData.a_tyUpstreamConfigurations[p_udiRmtIndexUS1].iUpstreamLaneId;
			tyConfigurationWr.a_tyUSParam[0].sHostAddress           	:= p_tyRmtSetConfiguration.tyData.a_tyUpstreamConfigurations[p_udiRmtIndexUS1].sHostAddress;
			tyConfigurationWr.a_tyUSParam[0].uiHostPort	                := p_tyRmtSetConfiguration.tyData.a_tyUpstreamConfigurations[p_udiRmtIndexUS1].uiPort;
			tyConfigurationWr.a_tyUSParam[0].sUpstreamInterfaceId   	:= p_tyRmtSetConfiguration.tyData.a_tyUpstreamConfigurations[p_udiRmtIndexUS1].sUpstreamInterfaceId;
		END_IF

		IF p_bRmtFoundIndexUS2 THEN
			tyConfigurationWr.a_tyUSParam[1].iLaneID		            := p_tyRmtSetConfiguration.tyData.a_tyUpstreamConfigurations[p_udiRmtIndexUS2].iUpstreamLaneId;
			tyConfigurationWr.a_tyUSParam[1].sHostAddress           	:= p_tyRmtSetConfiguration.tyData.a_tyUpstreamConfigurations[p_udiRmtIndexUS2].sHostAddress;
			tyConfigurationWr.a_tyUSParam[1].uiHostPort	                := p_tyRmtSetConfiguration.tyData.a_tyUpstreamConfigurations[p_udiRmtIndexUS2].uiPort;
			tyConfigurationWr.a_tyUSParam[1].sUpstreamInterfaceId   	:= p_tyRmtSetConfiguration.tyData.a_tyUpstreamConfigurations[p_udiRmtIndexUS2].sUpstreamInterfaceId;
		END_IF

		IF p_bRmtFoundIndexUS3 THEN
			tyConfigurationWr.a_tyUSParam[2].iLaneID		            := p_tyRmtSetConfiguration.tyData.a_tyUpstreamConfigurations[p_udiRmtIndexUS3].iUpstreamLaneId;
			tyConfigurationWr.a_tyUSParam[2].sHostAddress           	:= p_tyRmtSetConfiguration.tyData.a_tyUpstreamConfigurations[p_udiRmtIndexUS3].sHostAddress;
			tyConfigurationWr.a_tyUSParam[2].uiHostPort	                := p_tyRmtSetConfiguration.tyData.a_tyUpstreamConfigurations[p_udiRmtIndexUS3].uiPort;
			tyConfigurationWr.a_tyUSParam[2].sUpstreamInterfaceId   	:= p_tyRmtSetConfiguration.tyData.a_tyUpstreamConfigurations[p_udiRmtIndexUS3].sUpstreamInterfaceId;
		END_IF

		IF p_bRmtFoundIndexUS4 THEN
			tyConfigurationWr.a_tyUSParam[3].iLaneID		            := p_tyRmtSetConfiguration.tyData.a_tyUpstreamConfigurations[p_udiRmtIndexUS4].iUpstreamLaneId;
			tyConfigurationWr.a_tyUSParam[3].sHostAddress           	:= p_tyRmtSetConfiguration.tyData.a_tyUpstreamConfigurations[p_udiRmtIndexUS4].sHostAddress;
			tyConfigurationWr.a_tyUSParam[3].uiHostPort	                := p_tyRmtSetConfiguration.tyData.a_tyUpstreamConfigurations[p_udiRmtIndexUS4].uiPort;
			tyConfigurationWr.a_tyUSParam[3].sUpstreamInterfaceId   	:= p_tyRmtSetConfiguration.tyData.a_tyUpstreamConfigurations[p_udiRmtIndexUS4].sUpstreamInterfaceId;
		END_IF

		IF p_bRmtFoundIndexDS1 THEN
			tyConfigurationWr.a_tyDSParam[0].iLaneID	            	:= p_tyRmtSetConfiguration.tyData.a_tyDownstreamConfigurations[p_udiRmtIndexDS1].iDownstreamLaneId;
			tyConfigurationWr.a_tyDSParam[0].uiSvrPort               	:= p_tyRmtSetConfiguration.tyData.a_tyDownstreamConfigurations[p_udiRmtIndexDS1].uiPort;
			tyConfigurationWr.a_tyDSParam[0].sDownstreamInterfaceId  	:= p_tyRmtSetConfiguration.tyData.a_tyDownstreamConfigurations[p_udiRmtIndexDS1].sDownstreamInterfaceId;
		END_IF

		IF p_bRmtFoundIndexDS2 THEN
			tyConfigurationWr.a_tyDSParam[1].iLaneID	            	:= p_tyRmtSetConfiguration.tyData.a_tyDownstreamConfigurations[p_udiRmtIndexDS2].iDownstreamLaneId;
			tyConfigurationWr.a_tyDSParam[1].uiSvrPort               	:= p_tyRmtSetConfiguration.tyData.a_tyDownstreamConfigurations[p_udiRmtIndexDS2].uiPort;
			tyConfigurationWr.a_tyDSParam[1].sDownstreamInterfaceId  	:= p_tyRmtSetConfiguration.tyData.a_tyDownstreamConfigurations[p_udiRmtIndexDS2].sDownstreamInterfaceId;
		END_IF

		IF p_bRmtFoundIndexDS3 THEN
			tyConfigurationWr.a_tyDSParam[2].iLaneID	            	:= p_tyRmtSetConfiguration.tyData.a_tyDownstreamConfigurations[p_udiRmtIndexDS3].iDownstreamLaneId;
			tyConfigurationWr.a_tyDSParam[2].uiSvrPort               	:= p_tyRmtSetConfiguration.tyData.a_tyDownstreamConfigurations[p_udiRmtIndexDS3].uiPort;
			tyConfigurationWr.a_tyDSParam[2].sDownstreamInterfaceId  	:= p_tyRmtSetConfiguration.tyData.a_tyDownstreamConfigurations[p_udiRmtIndexDS3].sDownstreamInterfaceId;
		END_IF

		IF p_bRmtFoundIndexDS4 THEN
			tyConfigurationWr.a_tyDSParam[3].iLaneID	            	:= p_tyRmtSetConfiguration.tyData.a_tyDownstreamConfigurations[p_udiRmtIndexDS4].iDownstreamLaneId;
			tyConfigurationWr.a_tyDSParam[3].uiSvrPort               	:= p_tyRmtSetConfiguration.tyData.a_tyDownstreamConfigurations[p_udiRmtIndexDS4].uiPort;
			tyConfigurationWr.a_tyDSParam[3].sDownstreamInterfaceId  	:= p_tyRmtSetConfiguration.tyData.a_tyDownstreamConfigurations[p_udiRmtIndexDS4].sDownstreamInterfaceId;
		END_IF

		IF p_tyRmtSetConfiguration.tyAvl.bMachineId = TRUE THEN

			tyConfigurationWr.a_tyUSParam[0].sMachineId		:= p_tyRmtSetConfiguration.tyData.sMachineId;
			tyConfigurationWr.a_tyDSParam[0].sMachineId		:= p_tyRmtSetConfiguration.tyData.sMachineId;
			tyConfigurationWr.tySvyParam.sMachineId		    := p_tyRmtSetConfiguration.tyData.sMachineId;

		END_IF

		IF p_tyRmtSetConfiguration.tyAvl.bSupervisorySystemPort = TRUE THEN

			tyConfigurationWr.tySvyParam.uiSvySvstemPort	:= p_tyRmtSetConfiguration.tyData.uiSupervisorySystemPort;

		END_IF

	ELSIF p_bUISaveHMIConfigure THEN //Save US, DS Configure in HMI

	//	tyConfigurationWr.a_tyUSParam[0]  := pa_tyUSParam[0]; //lane 1 US
		tyConfigurationWr.a_tyDSParam[0]  := pa_tyDSParam[0]; //lane 1 DS
	//	tyConfigurationWr.a_tyUSParam[1]  := pa_tyUSParam[1]; //lane 2 US
		tyConfigurationWr.a_tyDSParam[1]  := pa_tyDSParam[1]; //lane 2 DS
	//	tyConfigurationWr.a_tyUSParam[2]  := pa_tyUSParam[2]; //lane 3 US
		tyConfigurationWr.a_tyDSParam[2]  := pa_tyDSParam[2]; //lane 3 DS
	//	tyConfigurationWr.a_tyUSParam[3]  := pa_tyUSParam[3]; //lane 4 US
		tyConfigurationWr.a_tyDSParam[3]  := pa_tyDSParam[3]; //lane 4 DS

	ELSIF p_bUISaveHMISvyConfig THEN //Save Supervisory Configure in HMI

		tyConfigurationWr.tySvyParam  := p_tySvyParam;

	END_IF

END_ACTION
```

#### Act_InitGlobal.st
```iecst
(** 2021-08-01 **)
ACTION Act_InitGlobal:

	(* Always Change If Project Change *)

	//Pass Data To Link
	p_bLinkStartupRun ACCESS p_StartupRun;
	pa_usiMacAddr ACCESS p_HWInfoMacAddr;
	p_tyDTStructure ACCESS p_TimeCurrDTStruct;

//	pa_tyLinkXMLTableDataBrdAvl1 ACCESS p_USHermesTableDataBrdAvl; //lane 1 B.A
//	p_iLinkXMLTableDataBrdAvlTtlIdx1 ACCESS p_USHermesTableDataBrdAvlTtlIdx; //lane 1 B.A
//	pa_tyLinkXMLTableDataBrdAvl2 ACCESS p_USHermesTableDataBrdAvl2; //lane 2 B.A
//	p_iLinkXMLTableDataBrdAvlTtlIdx2 ACCESS p_USHermesTableDataBrdAvlTtlIdx2; //lane 2 B.A
//	pa_tyLinkXMLTableDataBrdAvl3 ACCESS p_USHermesTableDataBrdAvl3; //lane 3 B.A
//	p_iLinkXMLTableDataBrdAvlTtlIdx3 ACCESS p_USHermesTableDataBrdAvlTtlIdx3; //lane 3 B.A
//	pa_tyLinkXMLTableDataBrdAvl4 ACCESS p_USHermesTableDataBrdAvl4; //lane 4 B.A
//	p_iLinkXMLTableDataBrdAvlTtlIdx4 ACCESS p_USHermesTableDataBrdAvlTtlIdx4; //lane 4 B.A
	p_bLinkOpsInitGConv1StepInitDone ACCESS p_OpsTravLifLDInitDone;
//	p_bLinkOpsInitGConv1MidHvBrd ACCESS p_OpsInitConvMidHvBrd;
//	p_bLinkOpsInitGConv1EndHvBrd ACCESS p_OpsInitConvEndHvBrd;
	p_bLinkOpsGConv1HvBrd ACCESS p_PullConvHvBrd;
//	p_bLinkUSHermesTransporting ACCESS p_USHermesTransporting;
//	p_bLinkUSSMEMATransporting ACCESS p_USSMEMATransporting;
	p_bLinkOpsGConv1StepEntBrd ACCESS p_OpsTravLifLDEntBrd;
//	p_bLinkOpsInitGConv2StepInitDone ACCESS p_OpsInitGConv2StepInitDone;  //Zone2
//	p_bLinkOpsInitGConv2MidHvBrd ACCESS p_OpsInitGConv2MidHvBrd;  //Zone2
//	p_bLinkOpsInitGConv2EndHvBrd ACCESS p_OpsInitGConv2EndHvBrd;  //Zone2
//	p_bLinkOpsGConv2HvBrd ACCESS p_OpsGConv2HvBrd;  //Zone2
//	p_bLinkOpsGConv2StepEntBrd ACCESS p_OpsGConv2StepEntBrd;  //Zone2
//	p_bLinkUSSMEMA2Transporting ACCESS p_USSMEMA2Transporting;  //Zone2

	//Pass Data To Internal Use
	p_udiRstErr ACCESS p_RstErrReset;
	p_bPrep ACCESS p_NtParamHermesPrep;
//	pa_tyUSParam ACCESS p_UIHermesUSParamWr; //HMI US Configure from UI
	pa_tyDSParam ACCESS p_UIHermesDSParamWr; //HMI DS Configure from UI
	p_tySvyParam ACCESS p_UIHermesSvyParamWr; //HMI Svy Configure from UI
	p_tyRmtSetConfiguration ACCESS p_RmtHermesSetConfiguration; //US,DS SetConfigure from RmtHermes
	p_tySvySetConfiguration ACCESS p_SvyHermesSetConfiguration; //US,DS SetConfigure from SvyHermes
	p_bRmtPrep ACCESS p_NtParamHermesRmtPrep;
	p_bRmtEn ACCESS p_McParamHermesRmtEn;
	p_bSvyPrep ACCESS p_NtParamHermesSvyPrep;
	p_bSvyEn ACCESS p_McParamHermesSvyEn;
	p_sRetainFileName1 ACCESS p_NtParamHermesRetainFileNm; //lane 1
//	p_sRetainFileName2 ACCESS p_NtParamHermesRetainFileNm2; //lane 2, rename to HermesL2.dat
//	p_sRetainFileName3 ACCESS p_NtParamHermesRetainFileNm3; //lane 3, rename to HermesL3.dat
//	p_sRetainFileName4 ACCESS p_NtParamHermesRetainFileNm4; //lane 4, rename to HermesL4.dat
	p_sConfigFileName ACCESS p_NtParamHermesConfigFileNm;
	p_sProgNm ACCESS p_NtParamHermesProgNm;
	p_bNtSettingsLoadDone ACCESS p_StartupNtSettingsLoadDone;
	p_bRmtHermesWriteConfig ACCESS p_RmtHermesWriteConfig;
	p_bSvyHermesWriteConfig ACCESS p_SvyHermesWriteConfig;
	p_bUISaveHMIConfigure ACCESS p_UISaveHMIConfigure;
	p_bUISaveHMISvyConfig ACCESS p_UISaveHMISvyConfig;
	p_sMcId ACCESS p_McParamMcNm;

	p_bRmtFoundIndexUS1 ACCESS p_RmtHermesFoundIndexUS1;
	p_bRmtFoundIndexUS2 ACCESS p_RmtHermesFoundIndexUS2;
	p_bRmtFoundIndexUS3 ACCESS p_RmtHermesFoundIndexUS3;
	p_bRmtFoundIndexUS4 ACCESS p_RmtHermesFoundIndexUS4;
	p_bRmtFoundIndexDS1 ACCESS p_RmtHermesFoundIndexDS1;
	p_bRmtFoundIndexDS2 ACCESS p_RmtHermesFoundIndexDS2;
	p_bRmtFoundIndexDS3 ACCESS p_RmtHermesFoundIndexDS3;
	p_bRmtFoundIndexDS4 ACCESS p_RmtHermesFoundIndexDS4;
	p_udiRmtIndexUS1 ACCESS p_RmtHermesIndexUS1;
	p_udiRmtIndexUS2 ACCESS p_RmtHermesIndexUS2;
	p_udiRmtIndexUS3 ACCESS p_RmtHermesIndexUS3;
	p_udiRmtIndexUS4 ACCESS p_RmtHermesIndexUS4;
	p_udiRmtIndexDS1 ACCESS p_RmtHermesIndexDS1;
	p_udiRmtIndexDS2 ACCESS p_RmtHermesIndexDS2;
	p_udiRmtIndexDS3 ACCESS p_RmtHermesIndexDS3;
	p_udiRmtIndexDS4 ACCESS p_RmtHermesIndexDS4;

	p_bSvyFoundIndexUS1 ACCESS p_SvyHermesFoundIndexUS1;
	p_bSvyFoundIndexUS2 ACCESS p_SvyHermesFoundIndexUS2;
	p_bSvyFoundIndexUS3 ACCESS p_SvyHermesFoundIndexUS3;
	p_bSvyFoundIndexUS4 ACCESS p_SvyHermesFoundIndexUS4;
	p_bSvyFoundIndexDS1 ACCESS p_SvyHermesFoundIndexDS1;
	p_bSvyFoundIndexDS2 ACCESS p_SvyHermesFoundIndexDS2;
	p_bSvyFoundIndexDS3 ACCESS p_SvyHermesFoundIndexDS3;
	p_bSvyFoundIndexDS4 ACCESS p_SvyHermesFoundIndexDS4;
	p_udiSvyIndexUS1 ACCESS p_SvyHermesIndexUS1;
	p_udiSvyIndexUS2 ACCESS p_SvyHermesIndexUS2;
	p_udiSvyIndexUS3 ACCESS p_SvyHermesIndexUS3;
	p_udiSvyIndexUS4 ACCESS p_SvyHermesIndexUS4;
	p_udiSvyIndexDS1 ACCESS p_SvyHermesIndexDS1;
	p_udiSvyIndexDS2 ACCESS p_SvyHermesIndexDS2;
	p_udiSvyIndexDS3 ACCESS p_SvyHermesIndexDS3;
	p_udiSvyIndexDS4 ACCESS p_SvyHermesIndexDS4;

	(* Always Change If Project Change *)
END_ACTION
```

#### Act_InitLocal.st
```iecst
(** 2021-08-01 **)
ACTION Act_InitLocal:

	//Input Reference Link To Local Variable
	p_eAct ACCESS ADR(eAct);
	p_udiRstErr ACCESS ADR(udiRstErr);
	p_bPrep ACCESS ADR(bPrep);
	p_bEn ACCESS ADR(bEn);
	p_bDis ACCESS ADR(bDis);
	pa_tyUSParam ACCESS ADR(a_tyUSParam);
	pa_tyDSParam ACCESS ADR(a_tyDSParam);
	p_tyRmtParam ACCESS ADR(tyRmtParam);
	p_tySvyParam ACCESS ADR(tySvyParam);
	p_tyRmtSetConfiguration ACCESS ADR(tyRmtSetConfiguration);
	p_tySvySetConfiguration ACCESS ADR(tySvySetConfiguration);
	p_bRmtPrep ACCESS ADR(bRmtPrep);
	p_bRmtEn ACCESS ADR(bRmtEn);
	p_bSvyPrep ACCESS ADR(bSvyPrep);
	p_bSvyEn ACCESS ADR(bSvyEn);
	p_sRetainFileName1 ACCESS ADR(sRetainFileName1);
	p_sRetainFileName2 ACCESS ADR(sRetainFileName2);
	p_sRetainFileName3 ACCESS ADR(sRetainFileName3);
	p_sRetainFileName4 ACCESS ADR(sRetainFileName4);
	p_udiRetainDataAddr1 ACCESS ADR(udiRetainDataAddr1);
	p_udiRetainDataLen1 ACCESS ADR(udiRetainDataLen1);
	p_udiRetainDataAddr2 ACCESS ADR(udiRetainDataAddr2);
	p_udiRetainDataLen2 ACCESS ADR(udiRetainDataLen2);
	p_udiRetainDataAddr3 ACCESS ADR(udiRetainDataAddr3);
	p_udiRetainDataLen3 ACCESS ADR(udiRetainDataLen3);
	p_udiRetainDataAddr4 ACCESS ADR(udiRetainDataAddr4);
	p_udiRetainDataLen4 ACCESS ADR(udiRetainDataLen4);
	p_sConfigFileName ACCESS ADR(sConfigFileName);
	p_sProgNm ACCESS ADR(sProgNm);
	p_bNtSettingsLoadDone ACCESS ADR(bNtSettingsLoadDone);
	p_bRmtHermesWriteConfig ACCESS ADR(bRmtHermesWriteConfig);
	p_bSvyHermesWriteConfig ACCESS ADR(bSvyHermesWriteConfig);
	p_bUISaveHMIConfigure ACCESS ADR(bUISaveHMIConfigure);
	p_bUISaveHMISvyConfig ACCESS ADR(bUISaveHMISvyConfig);
	p_sMcId ACCESS ADR(sMcId);

	p_bRmtFoundIndexUS1 ACCESS ADR(bRmtFoundIndexUS1);
	p_bRmtFoundIndexUS2 ACCESS ADR(bRmtFoundIndexUS2);
	p_bRmtFoundIndexUS3 ACCESS ADR(bRmtFoundIndexUS3);
	p_bRmtFoundIndexUS4 ACCESS ADR(bRmtFoundIndexUS4);
	p_bRmtFoundIndexDS1 ACCESS ADR(bRmtFoundIndexDS1);
	p_bRmtFoundIndexDS2 ACCESS ADR(bRmtFoundIndexDS2);
	p_bRmtFoundIndexDS3 ACCESS ADR(bRmtFoundIndexDS3);
	p_bRmtFoundIndexDS4 ACCESS ADR(bRmtFoundIndexDS4);
	p_udiRmtIndexUS1 ACCESS ADR(udiRmtIndexUS1);
	p_udiRmtIndexUS2 ACCESS ADR(udiRmtIndexUS2);
	p_udiRmtIndexUS3 ACCESS ADR(udiRmtIndexUS3);
	p_udiRmtIndexUS4 ACCESS ADR(udiRmtIndexUS4);
	p_udiRmtIndexDS1 ACCESS ADR(udiRmtIndexDS1);
	p_udiRmtIndexDS2 ACCESS ADR(udiRmtIndexDS2);
	p_udiRmtIndexDS3 ACCESS ADR(udiRmtIndexDS3);
	p_udiRmtIndexDS4 ACCESS ADR(udiRmtIndexDS4);

	p_bSvyFoundIndexUS1 ACCESS ADR(bSvyFoundIndexUS1);
	p_bSvyFoundIndexUS2 ACCESS ADR(bSvyFoundIndexUS2);
	p_bSvyFoundIndexUS3 ACCESS ADR(bSvyFoundIndexUS3);
	p_bSvyFoundIndexUS4 ACCESS ADR(bSvyFoundIndexUS4);
	p_bSvyFoundIndexDS1 ACCESS ADR(bSvyFoundIndexDS1);
	p_bSvyFoundIndexDS2 ACCESS ADR(bSvyFoundIndexDS2);
	p_bSvyFoundIndexDS3 ACCESS ADR(bSvyFoundIndexDS3);
	p_bSvyFoundIndexDS4 ACCESS ADR(bSvyFoundIndexDS4);
	p_udiSvyIndexUS1 ACCESS ADR(udiSvyIndexUS1);
	p_udiSvyIndexUS2 ACCESS ADR(udiSvyIndexUS2);
	p_udiSvyIndexUS3 ACCESS ADR(udiSvyIndexUS3);
	p_udiSvyIndexUS4 ACCESS ADR(udiSvyIndexUS4);
	p_udiSvyIndexDS1 ACCESS ADR(udiSvyIndexDS1);
	p_udiSvyIndexDS2 ACCESS ADR(udiSvyIndexDS2);
	p_udiSvyIndexDS3 ACCESS ADR(udiSvyIndexDS3);
	p_udiSvyIndexDS4 ACCESS ADR(udiSvyIndexDS4);

END_ACTION
```

#### Act_Link.st
```iecst
(** 2021-08-01 **)
ACTION Act_Link:

	//B.A Retain Data Lane 1
	p_udiRetainDataAddr1	:= ADR(a_tyHermesBrdAvlData);
	p_udiRetainDataLen1  	:= SIZEOF(a_tyHermesBrdAvlData);

	IF p_bLinkStartupRun = FALSE THEN

		//Passing Board Available Memory
		//Zone 1
		IF EDGEPOS(p_bLinkOpsInitGConv1StepInitDone) THEN

		//	IF (p_bLinkOpsInitGConv1MidHvBrd = FALSE) AND (p_bLinkOpsInitGConv1EndHvBrd = FALSE) THEN
				a_tyHermesBrdAvlData[1].bNewBrdAvl	:= TRUE;
				bHermesWriteRetainLane1					:= TRUE;
		//	END_IF

		END_IF

//		IF EDGEPOS(p_bLinkOpsGConv1HvBrd) AND (p_bLinkOpsGConv1StepEntBrd = TRUE) THEN
//
//			IF (p_bLinkUSHermesTransporting = TRUE) THEN
//				a_tyHermesBrdAvlData[1].a_tyXMLTableDataBrdAvl		:= pa_tyLinkXMLTableDataBrdAvl1;
//				a_tyHermesBrdAvlData[1].iXMLTableDataBrdAvlTtlIdx	:= p_iLinkXMLTableDataBrdAvlTtlIdx1;
//				a_tyHermesBrdAvlData[1].bNewBrdAvl					:= FALSE;
//				bHermesWriteRetainLane1									:= TRUE;
//			ELSE
//				a_tyHermesBrdAvlData[1].bNewBrdAvl	:= TRUE;
//				bHermesWriteRetainLane1					:= TRUE;
//			END_IF
//
//		END_IF
//
//		IF EDGENEG(p_bLinkOpsGConv1HvBrd) AND (p_bLinkOpsInitGConv1StepInitDone = TRUE) THEN
//			a_tyHermesBrdAvlData[1].bNewBrdAvl	:= TRUE;
//			bHermesWriteRetainLane1					:= TRUE;
//		END_IF

//		//Zone 2 get from Zone 1
//		IF EDGEPOS(p_bLinkOpsInitGConv2StepInitDone) THEN
//
//			IF (p_bLinkOpsInitGConv2MidHvBrd = FALSE) AND (p_bLinkOpsInitGConv2EndHvBrd = FALSE) THEN
//				a_tyHermesBrdAvlData[2].bNewBrdAvl	:= TRUE;
//				bHermesWriteRetainLane1					:= TRUE;
//			END_IF
//
//		END_IF
//
//		IF EDGEPOS(p_bLinkOpsGConv2HvBrd) AND (p_bLinkOpsGConv2StepEntBrd = TRUE) THEN
//
//			IF (p_bLinkUSSMEMA2Transporting = TRUE) THEN
//				a_tyHermesBrdAvlData[2]	:= a_tyHermesBrdAvlData[1];
//				bHermesWriteRetainLane1		:= TRUE;
//			ELSE
//				a_tyHermesBrdAvlData[2].bNewBrdAvl	:= TRUE;
//				bHermesWriteRetainLane1					:= TRUE;
		//			END_IF

//
//		END_IF
//
//		IF EDGENEG(p_bLinkOpsGConv2HvBrd) AND (p_bLinkOpsInitGConv2StepInitDone = TRUE) THEN
//			a_tyHermesBrdAvlData[2].bNewBrdAvl	:= TRUE;
//			bHermesWriteRetainLane1					:= TRUE;
//		END_IF

		//Zone 3 get from Zone 2 and so on. Duplicate if needed.

		//Write Hermes Retain Data
		IF bHermesWriteRetainLane1 = TRUE THEN
			p_eAct	:= HermesActWriteRetainLane1;

			IF (eStat = HermesActWriteRetainLane1) AND (eStatus = Done) THEN
				p_eAct				:= HermesActIdle;
				bHermesWriteRetainLane1	:= FALSE;
			END_IF

		END_IF

		IF EDGEPOS(p_bLinkOpsGConv1HvBrd) THEN
			fHermesGenerateUUID(ADR(sGenBrdUUID) , p_tyDTStructure , pa_usiMacAddr);
		END_IF

	//Dupplicate Lane 2 B.A data accordingly, make sure make condition where boolean bHermesWriteRetainLane1 must be false then only change p_eAct of Lane 2.

	END_IF

END_ACTION
```

#### Act_LinkAction.st
```iecst
(** 2021-08-01 **)
ACTION Act_LinkAction:

	IF p_bLinkStartupRun = TRUE THEN
		p_eAct ACCESS p_StartupHermesAct;
	ELSIF p_bSvyHermesWriteConfig THEN
		p_eAct ACCESS p_SvyHermesAct;
	ELSIF p_bRmtHermesWriteConfig THEN
		p_eAct ACCESS p_RmtHermesAct;
	ELSIF p_bUISaveHMIConfigure OR p_bUISaveHMISvyConfig THEN
		p_eAct ACCESS p_UIHermesAct;
	END_IF

END_ACTION
```

#### Init.st
```iecst
(** 2021-08-01 **)
PROGRAM _INIT

	(* Always Change If Project Change *)

	//Pass Address To Global Address For External Use
	//Action, State & Status
	p_HermesStat	:= ADR(eStat);
	p_HermesStatus	:= ADR(eStatus);
	p_HermesStatTxt	:= ADR(sStatTxt);

	//Alarm
	p_HermesAlmData	:= ADR(tyAlmData);

	//Output
	p_HermesFileNotFound	        	:= ADR(bFileNotFound);
	p_HermesConfiguration	        	:= ADR(tyCurrConfiguration);
	p_HermesConfigurationWr	        	:= ADR(tyConfigurationWr);
	p_HermesUSParam1		        	:= ADR(tyCurrConfiguration.a_tyUSParam[0]); //Lane 1
	p_HermesUSParam2	        		:= ADR(tyCurrConfiguration.a_tyUSParam[1]); //Lane 2
	p_HermesUSParam3		         	:= ADR(tyCurrConfiguration.a_tyUSParam[2]); //Lane 3
	p_HermesUSParam4		        	:= ADR(tyCurrConfiguration.a_tyUSParam[3]); //Lane 4
	p_HermesDSParam1		        	:= ADR(tyCurrConfiguration.a_tyDSParam[0]); //Lane 1
	p_HermesDSParam2		        	:= ADR(tyCurrConfiguration.a_tyDSParam[1]); //Lane 2
	p_HermesDSParam3		         	:= ADR(tyCurrConfiguration.a_tyDSParam[2]); //Lane 3
	p_HermesDSParam4		        	:= ADR(tyCurrConfiguration.a_tyDSParam[3]); //Lane 4
	p_HermesSvyParam		        	:= ADR(tyCurrConfiguration.tySvyParam);
	p_HermesBrdAvlDataTable1stZ		    := ADR(a_tyHermesBrdAvlData[1].a_tyXMLTableDataBrdAvl); //Lane 1 First Zone Data, for B.F
	p_HermesBrdAvlDataTtlIdx1stZ    	:= ADR(a_tyHermesBrdAvlData[1].iXMLTableDataBrdAvlTtlIdx);  //Lane 1 First Zone Data, for B.F
	p_HermesBrdAvlDataNewBrdAvl1stZ	    := ADR(a_tyHermesBrdAvlData[1].bNewBrdAvl);  //Lane 1 First Zone Data, for B.F
	p_HermesBrdAvlDataTableLastZ		:= ADR(a_tyHermesBrdAvlData[1].a_tyXMLTableDataBrdAvl); //Lane 1 Last Zone Data,for B.A, adjust array no. accordingly
	p_HermesBrdAvlDataTtlIdxLastZ	    := ADR(a_tyHermesBrdAvlData[1].iXMLTableDataBrdAvlTtlIdx); //Lane 1 Last Zone Data,for B.A, adjust array no. accordingly
	p_HermesBrdAvlDataNewBrdAvlLastZ	:= ADR(a_tyHermesBrdAvlData[1].bNewBrdAvl); //Lane 1 Last Zone Data,for B.A, adjust array no. accordingly
	p_HermesBrdId						:= ADR(sGenBrdUUID);

	(* Always Change If Project Change *)
END_PROGRAM
```

### DSHermesA.var - Change By Project
```iecst
(*2021-08-01*)
(**)
(*Action & State & Status*)
VAR
	p_DSHermesAStat : UDINT;
	p_DSHermesAStatus : UDINT;
	p_DSHermesAStatTxt : UDINT;
END_VAR
(**)
(*Alarm*)
VAR
	p_DSHermesAAlmData : UDINT;
	p_DSHermesAAlmData1 : UDINT;
	p_DSHermesAAlmData2 : UDINT;
	p_DSHermesAAlmData3 : UDINT;
	p_DSHermesAAlmData4 : UDINT;
END_VAR
(**)
(*Output*)
VAR
	p_DSHermesAFileNotFound : UDINT;
	p_DSHermesAConnected : UDINT;
	p_DSHermesAHandshakeDone : UDINT;
	p_DSHermesAUSRdy : UDINT;
	p_DSHermesADSRdy : UDINT;
	p_DSHermesAUSGdRdy : UDINT;
	p_DSHermesADSGdRdy : UDINT;
	p_DSHermesATransporting : UDINT;
	p_DSHermesAStopTransport : UDINT;
	p_DSHermesAInternalSnd : UDINT;
	p_DSHermesATransportFinishedSnd : UDINT;
	p_DSHermesABoardDepartedData : UDINT;
	p_DSHermesAAllZonesEmpty : UDINT;
	p_SendBFId : UDINT;
END_VAR
```

### Program Logical/Hermes/DSHermesA (IEC) - 1.00.0 - NtHermes v5.00.0 , NtTCP v5.00.0 , NtMessage v5.00.0

#### InputRef.var
```iecst
(*2021-08-01*)
(**)
(*General*)
VAR
	p_eAct : REFERENCE TO eHermesAction;
	p_udiRstErr : REFERENCE TO UDINT;
	p_bPrep : REFERENCE TO BOOL;
	p_bEn : REFERENCE TO BOOL;
	p_bDis : REFERENCE TO BOOL;
END_VAR
(**)
(*Configuration*)
VAR
	p_tyParam : REFERENCE TO tyHermesDSParam;
	p_sIPAddr : REFERENCE TO STRING[15];
	pa_usiMacAddr : REFERENCE TO ARRAY[0..5] OF USINT;
	p_tyDTStructure : REFERENCE TO DTStructure;
	p_dtCurrDT : REFERENCE TO DATE_AND_TIME;
	p_sMcId : REFERENCE TO STRING[80];
END_VAR
(**)
(*Input*)
VAR
	p_bRdySnd : REFERENCE TO BOOL;
	p_bSndCompl : REFERENCE TO BOOL;
	p_bSndIncompl : REFERENCE TO BOOL;
	p_bSndNotStart : REFERENCE TO BOOL;
	p_bBAWidthEn : REFERENCE TO BOOL; (*Board Available Check Width*)
	p_bBASltEn : REFERENCE TO BOOL; (*Board Available Check Slot*)
	p_bBFWidthEn : REFERENCE TO BOOL; (*Board Forecast Check Width*)
	p_bBFSltEn : REFERENCE TO BOOL; (*Board Forecast Check Slot*)
	p_sRecipeNm : REFERENCE TO STRING[254];
	p_sForecastId : REFERENCE TO STRING[80];
	p_sBoardId : REFERENCE TO STRING[36];
	p_sInterfaceId : REFERENCE TO STRING[80];
	p_sVersion : REFERENCE TO STRING[7];
	p_eFailedBoard : REFERENCE TO eHermesFailedBoard;
	p_eFlippedBoard : REFERENCE TO eHermesFlippedBoard;
	p_sTopBarcode : REFERENCE TO STRING[254];
	p_sBottomBarcode : REFERENCE TO STRING[254];
	p_rLength : REFERENCE TO REAL;
	p_rThickness : REFERENCE TO REAL;
	p_rConveyorSpeed : REFERENCE TO REAL;
	p_rTopClearanceHeight : REFERENCE TO REAL;
	p_rBottomClearanceHeight : REFERENCE TO REAL;
	p_rWeight : REFERENCE TO REAL;
	p_sWorkOrderId : REFERENCE TO STRING[80];
	p_sBatchId : REFERENCE TO STRING[80];
	p_diWidthInUM : REFERENCE TO DINT;
	p_diMinSltValue : REFERENCE TO DINT;
	p_diMaxSltValue : REFERENCE TO DINT;
	p_diPitch : REFERENCE TO DINT;
	p_diTtlSlt : REFERENCE TO DINT;
	p_diSltToSltInUM : REFERENCE TO DINT;
	p_udiSndBffrSize : REFERENCE TO UDINT;
	p_udiRcvBffrSize : REFERENCE TO UDINT;
	p_udiAliveIdleTimeInSec : REFERENCE TO UDINT;
	p_tConnTimeOut : REFERENCE TO TIME;
	p_diTransferInTO : REFERENCE TO DINT;
	pa_tyXMLTableDataBrdAvl : REFERENCE TO ARRAY[0..200] OF tyXMLTableDat;
	p_iXMLTableDataBrdAvlTtlIdx : REFERENCE TO INT;
	p_bNewBrdAvlFirstZone : REFERENCE TO BOOL;
	p_bNewBrdAvlLastZone : REFERENCE TO BOOL;
	p_bOpsRun : REFERENCE TO BOOL;
	p_bInterruptSen : REFERENCE TO BOOL;
	p_udiFileKeepDay : REFERENCE TO UDINT;
	p_udiRetainDataAddr : REFERENCE TO UDINT;
	p_udiRetainDataLen : REFERENCE TO UDINT;
	p_sRetainFileName : REFERENCE TO STRING[80];
	p_sProgNm : REFERENCE TO STRING[15];
	p_bNtSettingsLoadDone : REFERENCE TO BOOL;
	p_bRmtPrep : REFERENCE TO BOOL;
	p_bRmtEn : REFERENCE TO BOOL;
	p_bSvyPrep : REFERENCE TO BOOL;
	p_bSvyEn : REFERENCE TO BOOL;
	p_bOpsGConv1HvBrd : REFERENCE TO BOOL;
	p_bAllZonesEmpty : REFERENCE TO BOOL;
	p_bFirstZoneHaveBoard : REFERENCE TO BOOL;
	p_tyUSBoardArrivedData : REFERENCE TO tyHermesBoardAvailable;
	p_rMcCycleTm : REFERENCE TO REAL;
	p_rAWCycleTm : REFERENCE TO REAL;
	p_bInitDone : REFERENCE TO BOOL;
	p_tyHermesConfiguration : REFERENCE TO tyHermesConfiguration;
	p_bUSHermesStopTransport : REFERENCE TO BOOL;
	p_bRcvBoardInfo : REFERENCE TO BOOL;
	p_tyBoardInfoData : REFERENCE TO tyHermesSendBoardInfo;
	p_tySendWorkOrderData : REFERENCE TO tyHermesSendWorkOrderInfo;
	p_bUSHermesTransporting : REFERENCE TO BOOL;
	p_bReplyWorkOrderInfo : REFERENCE TO BOOL;
	p_bSendBoardForecast : REFERENCE TO BOOL;
	p_bClearWorkOrder : REFERENCE TO BOOL;
	p_bFirstZoneEndSen : REFERENCE TO BOOL;
	p_bNewProduct : REFERENCE TO BOOL;
	p_bNewWidth : REFERENCE TO BOOL;
	p_bInternalUse : REFERENCE TO BOOL;
	p_sInternalRcv : REFERENCE TO STRING[65535];
	p_tyDI : REFERENCE TO tyDigitalInput;
	p_eLinkCustomerReq : REFERENCE TO eCustomer;
	p_usiProdRcpCurrRcp1McMod : REFERENCE TO USINT;
	p_usiSelProdRcpStep : REFERENCE TO USINT;
END_VAR
(**)
(*Dummy*)
VAR
	p_sFoundAddressTop : REFERENCE TO STRING[254];
	p_sFoundAddressBottom : REFERENCE TO STRING[254];
END_VAR
```

#### InputRef_Link.var
```iecst
(*2021-08-01*)
(**)
VAR
	p_bLinkAWWidthPosDiff : REFERENCE TO BOOL;
	p_bLinkOpsAWStepMove : REFERENCE TO BOOL;
	p_bLinkProdRcpCurrAll : REFERENCE TO ARRAY[0..5] OF tyProdRcpParam;
END_VAR
(**)
VAR
	p_bLinkStartupRun : REFERENCE TO BOOL;
	p_eLinkMcParamDSCommMod : REFERENCE TO eMcSetCommMod;
	p_bLinkNtParamProjLaneBPrep : REFERENCE TO BOOL;
	bHermesRun : BOOL;
	bHermesStop : BOOL;
END_VAR
(**)
VAR
	p_usiLinkProdRcpCurrRcpFlipBrd : REFERENCE TO USINT;
	p_bLinkConvHvBrd : REFERENCE TO BOOL;
	p_bLinkOpsTravLifLDDSComm : REFERENCE TO BOOL;
	p_eLinkTravLifLDPosGo : REFERENCE TO eTravLifLDPos;
	p_tyAutoRcpTravLif : REFERENCE TO tyBoardProperty;
	p_diLinkAutoRcpTravLifWidth : REFERENCE TO DINT;
	p_diLinkAutoRcpMag1Width : REFERENCE TO DINT;
	p_diLinkAutoRcpMag2Width : REFERENCE TO DINT;
	p_diLinkAutoRcpMag3Width : REFERENCE TO DINT;
	p_tyAutoRcpMagRcp : REFERENCE TO ARRAY[1..4] OF tyBoardProperty;
	p_ausiSvyMagAccOrder : REFERENCE TO ARRAY[1..3] OF USINT;
	p_sHermesBrdId : REFERENCE TO STRING[36];
	p_bDIPullerRetRS : REFERENCE TO BOOL;
END_VAR
```
